C01822=1224.483,329.807,-70.540,-176.134,7.147,148.210
C01823=1224.479,330.055,-70.571,-176.132,7.149,148.210
C01824=1224.475,330.303,-70.602,-176.130,7.152,148.210
C01825=1224.470,330.551,-70.633,-176.128,7.155,148.211
C01826=1224.466,330.798,-70.664,-176.126,7.157,148.211
C01827=1224.462,331.047,-70.695,-176.124,7.160,148.211
C01828=1224.458,331.294,-70.727,-176.121,7.163,148.211
C01829=1224.454,331.543,-70.758,-176.120,7.165,148.211
C01830=1224.449,331.791,-70.789,-176.117,7.168,148.211
C01831=1224.445,332.039,-70.820,-176.115,7.171,148.211
C01832=1224.441,332.287,-70.851,-176.113,7.173,148.211
C01833=1224.436,332.535,-70.882,-176.111,7.176,148.211
C01834=1224.432,332.783,-70.914,-176.109,7.179,148.211
C01835=1224.428,333.031,-70.945,-176.107,7.181,148.211
C01836=1224.424,333.279,-70.976,-176.105,7.184,148.212
C01837=1224.419,333.527,-71.007,-176.103,7.187,148.212
C01838=1224.415,333.776,-71.038,-176.101,7.189,148.212
C01839=1224.411,334.023,-71.070,-176.099,7.192,148.212
C01840=1224.406,334.271,-71.101,-176.097,7.195,148.212
C01841=1224.403,334.519,-71.132,-176.095,7.198,148.212
C01842=1224.398,334.767,-71.163,-176.093,7.200,148.212
C01843=1224.394,335.015,-71.195,-176.091,7.203,148.212
C01844=1224.390,335.263,-71.226,-176.089,7.206,148.212
C01845=1224.386,335.511,-71.258,-176.087,7.209,148.213
C01846=1224.381,335.759,-71.288,-176.085,7.211,148.212
C01847=1224.378,336.007,-71.320,-176.083,7.214,148.213
C01848=1224.373,336.254,-71.352,-176.081,7.217,148.213
C01849=1224.369,336.503,-71.383,-176.079,7.219,148.213
C01850=1224.365,336.750,-71.414,-176.077,7.222,148.213
C01851=1224.361,336.999,-71.445,-176.075,7.225,148.213
C01852=1224.356,337.247,-71.478,-176.073,7.227,148.213
C01853=1224.352,337.495,-71.509,-176.071,7.230,148.213
C01854=1224.348,337.743,-71.540,-176.069,7.233,148.214
C01855=1224.344,337.991,-71.572,-176.067,7.235,148.214
C01856=1224.339,338.239,-71.603,-176.065,7.238,148.214
C01857=1224.336,338.487,-71.635,-176.063,7.241,148.214
C01858=1224.331,338.734,-71.666,-176.061,7.243,148.214
C01859=1224.327,338.983,-71.697,-176.059,7.247,148.214
C01860=1224.323,339.231,-71.730,-176.057,7.249,148.214
C01861=1224.319,339.478,-71.761,-176.055,7.251,148.214
C01862=1224.315,339.727,-71.792,-176.053,7.255,148.215
C01863=1224.310,339.974,-71.824,-176.051,7.257,148.215
C01864=1224.307,340.222,-71.856,-176.049,7.261,148.215
C01865=1224.302,340.470,-71.888,-176.047,7.263,148.215
C01866=1224.298,340.719,-71.919,-176.046,7.265,148.215
C01867=1224.293,340.996,-71.954,-176.043,7.269,148.215
C01868=1224.289,341.274,-71.990,-176.041,7.272,148.216
C01869=1224.283,341.552,-72.025,-176.039,7.274,148.216
C01870=1224.279,341.829,-72.061,-176.037,7.278,148.216
C01871=1224.275,342.077,-72.093,-176.035,7.280,148.216
C01872=1224.271,342.325,-72.124,-176.033,7.284,148.216
C01873=1224.266,342.573,-72.156,-176.031,7.286,148.216
C01874=1224.262,342.821,-72.188,-176.029,7.288,148.216
C01875=1224.258,343.069,-72.219,-176.027,7.292,148.217
C01876=1224.253,343.317,-72.252,-176.026,7.294,148.217
C01877=1224.250,343.565,-72.283,-176.024,7.297,148.217
C01878=1224.245,343.813,-72.315,-176.022,7.300,148.217
C01879=1224.242,344.061,-72.347,-176.020,7.302,148.217
C01880=1224.237,344.308,-72.379,-176.018,7.305,148.217
C01881=1224.233,344.557,-72.410,-176.016,7.308,148.218
C01882=1224.229,344.805,-72.442,-176.014,7.311,148.218
C01883=1224.224,345.053,-72.474,-176.013,7.313,148.218
C01884=1224.220,345.301,-72.506,-176.010,7.317,148.218
C01885=1224.216,345.549,-72.538,-176.009,7.319,148.218
C01886=1224.211,345.796,-72.570,-176.007,7.322,148.218
C01887=1224.208,346.044,-72.601,-176.005,7.325,148.219
C01888=1224.203,346.292,-72.634,-176.003,7.327,148.219
C01889=1224.199,346.540,-72.665,-176.001,7.330,148.219
C01890=1224.195,346.788,-72.697,-175.999,7.333,148.219
C01891=1224.190,347.036,-72.729,-175.997,7.336,148.219
C01892=1224.186,347.284,-72.761,-175.996,7.338,148.219
C01893=1224.182,347.532,-72.794,-175.994,7.341,148.220
C01894=1224.178,347.779,-72.825,-175.992,7.344,148.220
C01895=1224.174,348.027,-72.857,-175.990,7.347,148.220
C01896=1224.170,348.276,-72.889,-175.989,7.349,148.220
C01897=1224.166,348.523,-72.922,-175.987,7.352,148.220
C01898=1224.161,348.771,-72.954,-175.985,7.355,148.221
C01899=1224.157,349.019,-72.986,-175.983,7.357,148.221
C01900=1224.153,349.267,-73.018,-175.981,7.361,148.221
C01901=1224.149,349.515,-73.050,-175.979,7.363,148.221
C01902=1224.144,349.763,-73.082,-175.978,7.366,148.221
C01903=1224.141,350.011,-73.114,-175.976,7.368,148.222
C01904=1224.136,350.258,-73.146,-175.974,7.372,148.222
C01905=1224.132,350.506,-73.179,-175.972,7.374,148.222
C01906=1224.128,350.754,-73.211,-175.971,7.377,148.222
C01907=1224.124,351.002,-73.243,-175.969,7.380,148.222
C01908=1224.120,351.250,-73.274,-175.967,7.383,148.223
C01909=1224.115,351.498,-73.307,-175.965,7.385,148.223
C01910=1224.112,351.746,-73.339,-175.964,7.388,148.223
C01911=1224.107,351.994,-73.372,-175.961,7.391,148.223
C01912=1224.102,352.242,-73.404,-175.960,7.394,148.223
C01913=1224.099,352.490,-73.436,-175.959,7.397,148.224
C01914=1224.094,352.737,-73.469,-175.957,7.399,148.224
C01915=1224.091,352.985,-73.501,-175.955,7.402,148.224
C01916=1224.086,353.233,-73.533,-175.953,7.405,148.224
C01917=1224.082,353.481,-73.565,-175.952,7.407,148.225
C01918=1224.078,353.729,-73.598,-175.949,7.411,148.225
C01919=1224.074,353.977,-73.630,-175.948,7.413,148.225
C01920=1224.070,354.225,-73.662,-175.946,7.416,148.225
C01921=1224.065,354.472,-73.695,-175.945,7.419,148.226
C01922=1224.061,354.720,-73.727,-175.943,7.422,148.226
C01923=1224.057,354.969,-73.759,-175.941,7.425,148.226
C01924=1224.053,355.216,-73.792,-175.940,7.427,148.226
C01925=1224.049,355.464,-73.824,-175.938,7.430,148.226
C01926=1224.044,355.711,-73.857,-175.936,7.433,148.227
C01927=1224.041,355.959,-73.889,-175.935,7.436,148.227
C01928=1224.036,356.208,-73.921,-175.933,7.438,148.227
C01929=1224.032,356.455,-73.954,-175.931,7.441,148.227
C01930=1224.028,356.704,-73.986,-175.929,7.444,148.228
C01931=1224.024,356.951,-74.019,-175.928,7.447,148.228
C01932=1224.020,357.199,-74.051,-175.926,7.450,148.228
C01933=1224.016,357.446,-74.084,-175.925,7.452,148.228
C01934=1224.011,357.695,-74.117,-175.923,7.455,148.229
C01935=1224.008,357.942,-74.149,-175.921,7.458,148.229
C01936=1224.003,358.190,-74.182,-175.920,7.461,148.229
C01937=1223.999,358.437,-74.214,-175.918,7.463,148.229
C01938=1223.994,358.686,-74.247,-175.916,7.466,148.230
C01939=1223.991,358.933,-74.279,-175.915,7.470,148.230
C01940=1223.986,359.182,-74.312,-175.913,7.472,148.230
C01941=1223.982,359.429,-74.345,-175.911,7.475,148.230
C01942=1223.979,359.677,-74.377,-175.910,7.477,148.231
C01943=1223.974,359.925,-74.410,-175.909,7.480,148.231
C01944=1223.970,360.173,-74.442,-175.906,7.483,148.231
C01945=1223.965,360.420,-74.475,-175.905,7.486,148.232
C01946=1223.961,360.669,-74.507,-175.904,7.489,148.232
C01947=1223.957,360.916,-74.540,-175.902,7.491,148.232
C01948=1223.953,361.164,-74.573,-175.901,7.494,148.232
C01949=1223.949,361.412,-74.606,-175.899,7.497,148.233
C01950=1223.945,361.660,-74.638,-175.897,7.500,148.233
C01951=1223.941,361.907,-74.671,-175.896,7.503,148.233
C01952=1223.937,362.156,-74.704,-175.894,7.505,148.233
C01953=1223.933,362.404,-74.737,-175.893,7.508,148.234
C01954=1223.929,362.651,-74.770,-175.891,7.511,148.234
C01955=1223.924,362.899,-74.802,-175.890,7.514,148.234
C01956=1223.920,363.146,-74.835,-175.888,7.517,148.235
C01957=1223.916,363.394,-74.868,-175.887,7.520,148.235
C01958=1223.911,363.642,-74.900,-175.885,7.522,148.235
C01959=1223.907,363.890,-74.934,-175.884,7.525,148.236
C01960=1223.904,364.138,-74.966,-175.882,7.528,148.236
C01961=1223.900,364.385,-74.999,-175.881,7.531,148.236
C01962=1223.895,364.634,-75.032,-175.879,7.534,148.236
C01963=1223.891,364.881,-75.065,-175.878,7.536,148.237
C01964=1223.887,365.129,-75.098,-175.876,7.539,148.237
C01965=1223.883,365.377,-75.131,-175.875,7.542,148.237
C01966=1223.879,365.625,-75.163,-175.873,7.544,148.237
C01967=1223.875,365.873,-75.196,-175.872,7.547,148.238
C01968=1223.871,366.120,-75.229,-175.870,7.551,148.238
C01969=1223.867,366.368,-75.263,-175.869,7.553,148.239
C01970=1223.863,366.616,-75.296,-175.867,7.556,148.239
C01971=1223.858,366.896,-75.333,-175.866,7.559,148.239
C01972=1223.853,367.176,-75.370,-175.864,7.562,148.240
C01973=1223.849,367.455,-75.408,-175.863,7.565,148.240
C01974=1223.844,367.735,-75.444,-175.861,7.569,148.240
C01975=1223.840,367.983,-75.478,-175.860,7.571,148.241
C01976=1223.836,368.231,-75.510,-175.858,7.574,148.241
C01977=1223.832,368.478,-75.543,-175.857,7.577,148.241
C01978=1223.828,368.726,-75.576,-175.856,7.580,148.242
C01979=1223.824,368.974,-75.610,-175.854,7.582,148.242
C01980=1223.820,369.221,-75.643,-175.853,7.585,148.242
C01981=1223.815,369.469,-75.676,-175.852,7.588,148.243
C01982=1223.811,369.717,-75.709,-175.850,7.590,148.243
C01983=1223.807,369.965,-75.742,-175.849,7.593,148.243
C01984=1223.803,370.212,-75.775,-175.848,7.596,148.244
C01985=1223.799,370.461,-75.808,-175.846,7.598,148.244
C01986=1223.794,370.708,-75.841,-175.845,7.602,148.244
C01987=1223.790,370.956,-75.874,-175.843,7.605,148.245
C01988=1223.786,371.204,-75.907,-175.842,7.607,148.245
C01989=1223.782,371.452,-75.940,-175.841,7.610,148.245
C01990=1223.778,371.699,-75.974,-175.839,7.613,148.246
C01991=1223.774,371.947,-76.007,-175.838,7.616,148.246
C01992=1223.770,372.194,-76.041,-175.837,7.618,148.246
C01993=1223.766,372.442,-76.074,-175.835,7.621,148.247
C01994=1223.762,372.690,-76.107,-175.834,7.624,148.247
C01995=1223.758,372.937,-76.140,-175.833,7.627,148.247
C01996=1223.753,373.185,-76.173,-175.832,7.630,148.248
C01997=1223.748,373.433,-76.207,-175.830,7.632,148.248
C01998=1223.744,373.681,-76.240,-175.829,7.635,148.248
C01999=1223.740,373.929,-76.273,-175.828,7.637,148.249
C02000=1223.736,374.176,-76.306,-175.827,7.640,148.249
C02001=1223.733,374.425,-76.340,-175.826,7.643,148.249
C02002=1223.728,374.672,-76.373,-175.825,7.645,148.250
C02003=1223.724,374.920,-76.406,-175.823,7.648,148.250
C02004=1223.720,375.167,-76.440,-175.822,7.651,148.250
C02005=1223.716,375.415,-76.473,-175.821,7.654,148.251
C02006=1223.712,375.663,-76.506,-175.820,7.656,148.251
C02007=1223.708,375.911,-76.540,-175.819,7.659,148.252
C02008=1223.704,376.158,-76.573,-175.817,7.662,148.252
C02009=1223.699,376.406,-76.607,-175.816,7.665,148.252
C02010=1223.695,376.653,-76.640,-175.815,7.668,148.253
C02011=1223.692,376.902,-76.674,-175.813,7.670,148.253
C02012=1223.687,377.150,-76.707,-175.812,7.673,148.253
C02013=1223.683,377.397,-76.740,-175.812,7.675,148.254
C02014=1223.679,377.645,-76.773,-175.810,7.678,148.254
C02015=1223.675,377.892,-76.807,-175.809,7.681,148.255
C02016=1223.671,378.140,-76.841,-175.808,7.684,148.255
C02017=1223.666,378.388,-76.874,-175.807,7.686,148.255
C02018=1223.662,378.636,-76.907,-175.806,7.689,148.256
C02019=1223.658,378.883,-76.941,-175.805,7.692,148.256
C02020=1223.655,379.131,-76.975,-175.803,7.695,148.257
C02021=1223.651,379.379,-77.008,-175.803,7.697,148.257
C02022=1223.646,379.626,-77.042,-175.802,7.700,148.257
C02023=1223.642,379.874,-77.075,-175.800,7.702,148.258
C02024=1223.638,380.122,-77.109,-175.799,7.705,148.258
C02025=1223.634,380.369,-77.142,-175.798,7.708,148.258
C02026=1223.629,380.617,-77.176,-175.797,7.711,148.259
C02027=1223.626,380.865,-77.210,-175.796,7.713,148.259
C02028=1223.622,381.113,-77.243,-175.795,7.716,148.260
C02029=1223.618,381.360,-77.277,-175.794,7.719,148.260
C02030=1223.614,381.608,-77.310,-175.793,7.721,148.260
C02031=1223.609,381.855,-77.344,-175.792,7.724,148.261
C02032=1223.605,382.103,-77.378,-175.791,7.726,148.261
C02033=1223.601,382.351,-77.411,-175.790,7.729,148.261
C02034=1223.597,382.599,-77.445,-175.789,7.732,148.262
C02035=1223.593,382.847,-77.479,-175.788,7.735,148.262
C02036=1223.588,383.094,-77.512,-175.787,7.737,148.263
C02037=1223.585,383.341,-77.546,-175.786,7.740,148.263
C02038=1223.580,383.590,-77.580,-175.785,7.743,148.264
C02039=1223.577,383.837,-77.614,-175.784,7.745,148.264
C02040=1223.572,384.085,-77.647,-175.783,7.747,148.264
C02041=1223.569,384.332,-77.681,-175.782,7.750,148.265
C02042=1223.564,384.580,-77.715,-175.781,7.753,148.265
C02043=1223.560,384.828,-77.749,-175.780,7.756,148.266
C02044=1223.556,385.076,-77.782,-175.779,7.758,148.266
C02045=1223.551,385.324,-77.816,-175.778,7.761,148.267
C02046=1223.548,385.571,-77.850,-175.777,7.764,148.267
C02047=1223.543,385.819,-77.883,-175.776,7.766,148.267
C02048=1223.539,386.067,-77.918,-175.775,7.768,148.268
C02049=1223.535,386.314,-77.951,-175.774,7.771,148.268
C02050=1223.532,386.562,-77.985,-175.773,7.774,148.268
C02051=1223.527,386.809,-78.019,-175.773,7.776,148.269
C02052=1223.523,387.057,-78.052,-175.771,7.779,148.269
C02053=1223.520,387.305,-78.086,-175.770,7.782,148.270
C02054=1223.515,387.553,-78.120,-175.770,7.784,148.270
C02055=1223.511,387.800,-78.154,-175.768,7.787,148.271
C02056=1223.507,388.047,-78.187,-175.768,7.790,148.271
C02057=1223.503,388.296,-78.222,-175.767,7.792,148.271
C02058=1223.499,388.543,-78.255,-175.766,7.795,148.272
C02059=1223.495,388.790,-78.289,-175.765,7.798,148.272
C02060=1223.490,389.038,-78.324,-175.764,7.800,148.273
C02061=1223.487,389.286,-78.357,-175.763,7.803,148.273
C02062=1223.482,389.534,-78.392,-175.763,7.805,148.274
C02063=1223.478,389.781,-78.425,-175.762,7.807,148.274
C02064=1223.474,390.028,-78.459,-175.760,7.810,148.274
C02065=1223.470,390.277,-78.493,-175.760,7.812,148.275
C02066=1223.466,390.524,-78.527,-175.759,7.815,148.275
C02067=1223.461,390.772,-78.561,-175.758,7.817,148.276
C02068=1223.458,391.020,-78.595,-175.757,7.820,148.276
C02069=1223.454,391.267,-78.628,-175.756,7.823,148.276
C02070=1223.450,391.515,-78.663,-175.756,7.825,148.277
C02071=1223.446,391.762,-78.697,-175.755,7.828,148.277
C02072=1223.441,392.011,-78.731,-175.754,7.830,148.278
C02073=1223.438,392.258,-78.765,-175.753,7.833,148.278
C02074=1223.433,392.505,-78.799,-175.753,7.835,148.279
C02075=1223.429,392.787,-78.837,-175.752,7.838,148.279
C02076=1223.424,393.068,-78.876,-175.751,7.841,148.280
C02077=1223.419,393.351,-78.915,-175.750,7.844,148.280
C02078=1223.415,393.632,-78.954,-175.749,7.847,148.281
C02079=1223.411,393.879,-78.988,-175.748,7.849,148.281
C02080=1223.406,394.127,-79.021,-175.747,7.852,148.281
C02081=1223.402,394.375,-79.056,-175.746,7.854,148.282
C02082=1223.399,394.622,-79.090,-175.746,7.857,148.282
C02083=1223.394,394.870,-79.125,-175.745,7.859,148.283
C02084=1223.390,395.118,-79.158,-175.744,7.862,148.283
C02085=1223.386,395.366,-79.193,-175.744,7.864,148.284
C02086=1223.382,395.613,-79.226,-175.743,7.867,148.284
C02087=1223.378,395.861,-79.261,-175.742,7.869,148.284
C02088=1223.374,396.109,-79.294,-175.741,7.872,148.285
C02089=1223.369,396.356,-79.329,-175.741,7.874,148.285
C02090=1223.366,396.604,-79.363,-175.739,7.877,148.286
C02091=1223.362,396.851,-79.398,-175.739,7.879,148.286
C02092=1223.358,397.098,-79.431,-175.738,7.882,148.287
C02093=1223.354,397.346,-79.466,-175.737,7.884,148.287
C02094=1223.350,397.594,-79.499,-175.737,7.886,148.288
C02095=1223.345,397.842,-79.534,-175.736,7.889,148.288
C02096=1223.342,398.089,-79.568,-175.735,7.891,148.288
C02097=1223.337,398.337,-79.603,-175.735,7.894,148.289
C02098=1223.333,398.584,-79.636,-175.734,7.896,148.289
C02099=1223.329,398.832,-79.671,-175.733,7.898,148.290
C02100=1223.325,399.080,-79.705,-175.733,7.901,148.290
C02101=1223.321,399.327,-79.739,-175.732,7.903,148.290
C02102=1223.317,399.575,-79.774,-175.731,7.906,148.291
C02103=1223.313,399.822,-79.808,-175.731,7.908,148.291
C02104=1223.309,400.071,-79.842,-175.730,7.910,148.292
C02105=1223.305,400.318,-79.876,-175.729,7.913,148.292
C02106=1223.301,400.565,-79.911,-175.729,7.915,148.293
C02107=1223.297,400.813,-79.946,-175.728,7.917,148.293
C02108=1223.293,401.060,-79.980,-175.727,7.920,148.294
C02109=1223.288,401.308,-80.014,-175.727,7.922,148.294
C02110=1223.285,401.556,-80.048,-175.725,7.925,148.294
C02111=1223.280,401.803,-80.083,-175.725,7.927,148.295
C02112=1223.276,402.052,-80.117,-175.725,7.929,148.295
C02113=1223.272,402.299,-80.151,-175.723,7.932,148.296
C02114=1223.268,402.546,-80.185,-175.723,7.934,148.296
C02115=1223.265,402.794,-80.219,-175.723,7.936,148.297
C02116=1223.260,403.041,-80.254,-175.722,7.939,148.297
C02117=1223.256,403.290,-80.289,-175.721,7.941,148.297
C02118=1223.252,403.537,-80.323,-175.721,7.943,148.298
C02119=1223.248,403.784,-80.357,-175.720,7.946,148.298
C02120=1223.244,404.032,-80.392,-175.719,7.949,148.299
C02121=1223.240,404.279,-80.426,-175.719,7.950,148.299
C02122=1223.236,404.527,-80.461,-175.718,7.953,148.300
C02123=1223.231,404.775,-80.495,-175.718,7.955,148.300
C02124=1223.227,405.022,-80.529,-175.717,7.958,148.301
C02125=1223.223,405.270,-80.564,-175.716,7.960,148.301
C02126=1223.219,405.518,-80.598,-175.716,7.962,148.301
C02127=1223.216,405.765,-80.633,-175.715,7.965,148.302
C02128=1223.211,406.012,-80.668,-175.714,7.967,148.302
C02129=1223.207,406.260,-80.702,-175.714,7.969,148.303
C02130=1223.204,406.507,-80.736,-175.714,7.971,148.303
C02131=1223.199,406.755,-80.771,-175.712,7.974,148.303
C02132=1223.195,407.003,-80.806,-175.712,7.976,148.304
C02133=1223.191,407.250,-80.839,-175.712,7.978,148.304
C02134=1223.187,407.498,-80.874,-175.711,7.980,148.305
C02135=1223.183,407.746,-80.909,-175.711,7.982,148.305
C02136=1223.179,407.993,-80.943,-175.710,7.985,148.306
C02137=1223.175,408.241,-80.977,-175.709,7.988,148.306
C02138=1223.170,408.488,-81.012,-175.709,7.990,148.307
C02139=1223.167,408.736,-81.047,-175.708,7.992,148.307
C02140=1223.163,408.983,-81.081,-175.708,7.994,148.307
C02141=1223.159,409.231,-81.116,-175.707,7.997,148.308
C02142=1223.154,409.478,-81.151,-175.707,7.999,148.308
C02143=1223.151,409.726,-81.185,-175.706,8.001,148.309
C02144=1223.146,409.974,-81.219,-175.705,8.003,148.309
C02145=1223.143,410.222,-81.254,-175.705,8.005,148.310
C02146=1223.138,410.468,-81.289,-175.704,8.008,148.310
C02147=1223.135,410.716,-81.324,-175.704,8.010,148.311
C02148=1223.130,410.964,-81.358,-175.703,8.012,148.311
C02149=1223.126,411.211,-81.393,-175.702,8.014,148.311
C02150=1223.122,411.459,-81.427,-175.702,8.016,148.312
C02151=1223.118,411.706,-81.461,-175.702,8.018,148.312
C02152=1223.114,411.954,-81.497,-175.701,8.020,148.312
C02153=1223.110,412.201,-81.531,-175.700,8.023,148.313
C02154=1223.106,412.449,-81.566,-175.700,8.025,148.313
C02155=1223.102,412.697,-81.600,-175.699,8.028,148.314
C02156=1223.098,412.945,-81.635,-175.699,8.030,148.314
C02157=1223.094,413.191,-81.670,-175.698,8.032,148.315
C02158=1223.090,413.440,-81.705,-175.698,8.034,148.315
C02159=1223.086,413.687,-81.739,-175.697,8.036,148.315
C02160=1223.082,413.935,-81.774,-175.697,8.038,148.316
C02161=1223.078,414.182,-81.809,-175.696,8.041,148.316
C02162=1223.074,414.430,-81.844,-175.695,8.043,148.317
C02163=1223.069,414.677,-81.878,-175.695,8.045,148.317
C02164=1223.066,414.925,-81.912,-175.694,8.047,148.318
C02165=1223.062,415.172,-81.947,-175.694,8.049,148.318
C02166=1223.058,415.420,-81.982,-175.694,8.051,148.318
C02167=1223.051,415.838,-82.041,-175.692,8.055,148.319
C02168=1223.043,416.255,-82.099,-175.692,8.059,148.320
C02169=1223.037,416.673,-82.158,-175.691,8.063,148.321
C02170=1223.033,417.091,-82.216,-175.690,8.066,148.321
C02171=1222.612,417.091,-82.251,-175.693,8.076,148.325
C02172=1222.612,416.881,-82.221,-175.694,8.074,148.324
C02173=1222.615,416.671,-82.192,-175.694,8.073,148.324
C02174=1222.619,416.460,-82.162,-175.694,8.071,148.324
C02175=1222.622,416.250,-82.133,-175.695,8.069,148.324
C02176=1222.626,416.040,-82.103,-175.696,8.067,148.323
C02177=1222.628,415.830,-82.073,-175.696,8.065,148.323
C02178=1222.633,415.620,-82.044,-175.696,8.064,148.322
C02179=1222.635,415.409,-82.015,-175.697,8.062,148.322
C02180=1222.640,415.162,-81.980,-175.697,8.060,148.322
C02181=1222.644,414.914,-81.945,-175.697,8.058,148.321
C02182=1222.647,414.667,-81.911,-175.698,8.056,148.321
C02183=1222.651,414.419,-81.876,-175.699,8.054,148.320
C02184=1222.656,414.171,-81.841,-175.699,8.050,148.320
C02185=1222.660,413.924,-81.806,-175.700,8.049,148.320
C02186=1222.664,413.676,-81.771,-175.701,8.047,148.319
C02187=1222.667,413.429,-81.737,-175.701,8.044,148.319
C02188=1222.672,413.181,-81.703,-175.702,8.042,148.318
C02189=1222.676,412.934,-81.667,-175.702,8.040,148.318
C02190=1222.680,412.686,-81.633,-175.702,8.038,148.317
C02191=1222.684,412.438,-81.598,-175.703,8.036,148.317
C02192=1222.688,412.191,-81.564,-175.703,8.034,148.317
C02193=1222.692,411.943,-81.529,-175.704,8.031,148.316
C02194=1222.696,411.696,-81.494,-175.705,8.029,148.316
C02195=1222.700,411.448,-81.459,-175.705,8.027,148.315
C02196=1222.704,411.201,-81.425,-175.706,8.025,148.315
C02197=1222.709,410.954,-81.391,-175.706,8.022,148.314
C02198=1222.713,410.705,-81.356,-175.707,8.021,148.314
C02199=1222.717,410.459,-81.321,-175.708,8.018,148.314
C02200=1222.720,410.211,-81.286,-175.708,8.015,148.313
C02201=1222.725,409.963,-81.252,-175.709,8.013,148.313
C02202=1222.729,409.715,-81.217,-175.709,8.011,148.312
C02203=1222.733,409.468,-81.183,-175.710,8.009,148.312
C02204=1222.736,409.220,-81.148,-175.710,8.007,148.312
C02205=1222.741,408.973,-81.113,-175.711,8.004,148.311
C02206=1222.745,408.725,-81.078,-175.712,8.002,148.311
C02207=1222.749,408.478,-81.045,-175.712,8.000,148.310
C02208=1222.752,408.230,-81.010,-175.712,7.998,148.310
C02209=1222.757,407.982,-80.975,-175.713,7.996,148.309
C02210=1222.762,407.735,-80.941,-175.714,7.993,148.309
C02211=1222.765,407.487,-80.907,-175.714,7.991,148.308
C02212=1222.769,407.240,-80.872,-175.715,7.989,148.308
C02213=1222.773,406.992,-80.837,-175.715,7.987,148.308
C02214=1222.777,406.745,-80.803,-175.716,7.985,148.307
C02215=1222.781,406.497,-80.768,-175.717,7.981,148.307
C02216=1222.785,406.250,-80.733,-175.717,7.980,148.306
C02217=1222.789,406.003,-80.700,-175.717,7.977,148.306
C02218=1222.793,405.754,-80.665,-175.718,7.975,148.305
C02219=1222.798,405.507,-80.630,-175.719,7.972,148.305
C02220=1222.801,405.259,-80.596,-175.719,7.970,148.305
C02221=1222.806,405.012,-80.562,-175.720,7.968,148.304
C02222=1222.810,404.764,-80.527,-175.721,7.965,148.304
C02223=1222.813,404.517,-80.493,-175.721,7.963,148.303
C02224=1222.818,404.269,-80.458,-175.722,7.961,148.303
C02225=1222.822,404.021,-80.424,-175.722,7.959,148.302
C02226=1222.826,403.774,-80.390,-175.723,7.956,148.302
C02227=1222.830,403.526,-80.355,-175.724,7.954,148.301
C02228=1222.834,403.278,-80.320,-175.724,7.952,148.301
C02229=1222.838,403.031,-80.286,-175.725,7.949,148.301
C02230=1222.842,402.783,-80.252,-175.726,7.947,148.300
C02231=1222.847,402.536,-80.217,-175.726,7.945,148.300
C02232=1222.850,402.288,-80.183,-175.727,7.943,148.299
C02233=1222.855,402.040,-80.148,-175.728,7.940,148.299
C02234=1222.858,401.793,-80.115,-175.728,7.938,148.299
C02235=1222.862,401.545,-80.080,-175.728,7.935,148.298
C02236=1222.867,401.298,-80.045,-175.730,7.933,148.298
C02237=1222.870,401.050,-80.011,-175.730,7.931,148.297
C02238=1222.875,400.803,-79.977,-175.731,7.927,148.297
C02239=1222.879,400.555,-79.943,-175.732,7.926,148.296
C02240=1222.882,400.307,-79.908,-175.732,7.924,148.296
C02241=1222.887,400.059,-79.874,-175.733,7.920,148.295
C02242=1222.891,399.812,-79.840,-175.734,7.918,148.295
C02243=1222.895,399.564,-79.805,-175.734,7.916,148.294
C02244=1222.899,399.317,-79.772,-175.735,7.913,148.294
C02245=1222.903,399.069,-79.737,-175.736,7.911,148.294
C02246=1222.908,398.821,-79.702,-175.736,7.908,148.293
C02247=1222.911,398.574,-79.668,-175.737,7.906,148.293
C02248=1222.915,398.326,-79.634,-175.738,7.904,148.292
C02249=1222.919,398.079,-79.600,-175.738,7.901,148.292
C02250=1222.924,397.831,-79.566,-175.739,7.899,148.292
C02251=1222.927,397.583,-79.532,-175.740,7.896,148.291
C02252=1222.932,397.336,-79.497,-175.740,7.894,148.291
C02253=1222.936,397.089,-79.463,-175.741,7.892,148.290
C02254=1222.940,396.841,-79.429,-175.742,7.889,148.290
C02255=1222.943,396.593,-79.395,-175.742,7.887,148.289
C02256=1222.948,396.345,-79.361,-175.744,7.884,148.289
C02257=1222.952,396.097,-79.326,-175.744,7.882,148.289
C02258=1222.956,395.850,-79.292,-175.745,7.879,148.288
C02259=1222.961,395.603,-79.258,-175.746,7.877,148.288
C02260=1222.964,395.355,-79.224,-175.747,7.874,148.287
C02261=1222.969,395.107,-79.190,-175.747,7.872,148.287
C02262=1222.973,394.860,-79.156,-175.748,7.869,148.286
C02263=1222.977,394.612,-79.121,-175.749,7.867,148.286
C02264=1222.980,394.365,-79.087,-175.749,7.864,148.285
C02265=1222.985,394.117,-79.053,-175.750,7.862,148.285
C02266=1222.989,393.869,-79.019,-175.751,7.859,148.285
C02267=1222.992,393.622,-78.985,-175.751,7.857,148.284
C02268=1222.997,393.340,-78.946,-175.753,7.854,148.284
C02269=1223.002,393.058,-78.908,-175.753,7.851,148.283
C02270=1223.007,392.776,-78.868,-175.755,7.848,148.283
C02271=1223.011,392.494,-78.830,-175.755,7.845,148.282
C02272=1223.016,392.247,-78.796,-175.756,7.843,148.282
C02273=1223.019,392.000,-78.762,-175.757,7.840,148.281
C02274=1223.024,391.752,-78.729,-175.758,7.838,148.281
C02275=1223.028,391.504,-78.694,-175.758,7.835,148.280
C02276=1223.031,391.257,-78.660,-175.759,7.833,148.280
C02277=1223.036,391.009,-78.626,-175.760,7.831,148.280
C02278=1223.039,390.761,-78.592,-175.761,7.828,148.279
C02279=1223.044,390.514,-78.557,-175.762,7.825,148.279
C02280=1223.048,390.266,-78.524,-175.763,7.823,148.278
C02281=1223.052,390.019,-78.490,-175.763,7.821,148.278
C02282=1223.056,389.771,-78.456,-175.765,7.818,148.278
C02283=1223.060,389.523,-78.422,-175.765,7.815,148.277
C02284=1223.065,389.276,-78.388,-175.766,7.813,148.277
C02285=1223.069,389.028,-78.355,-175.767,7.810,148.276
C02286=1223.072,388.780,-78.321,-175.768,7.807,148.276
C02287=1223.077,388.533,-78.286,-175.769,7.805,148.275
C02288=1223.081,388.285,-78.253,-175.770,7.802,148.275
C02289=1223.085,388.038,-78.219,-175.770,7.800,148.275
C02290=1223.089,387.789,-78.185,-175.772,7.797,148.274
C02291=1223.093,387.542,-78.151,-175.773,7.794,148.274
C02292=1223.098,387.294,-78.117,-175.773,7.792,148.273
C02293=1223.101,387.047,-78.084,-175.774,7.789,148.273
C02294=1223.105,386.799,-78.049,-175.775,7.786,148.272
C02295=1223.110,386.551,-78.016,-175.776,7.784,148.272
C02296=1223.113,386.304,-77.982,-175.777,7.782,148.272
C02297=1223.118,386.056,-77.949,-175.778,7.779,148.271
C02298=1223.121,385.808,-77.914,-175.779,7.776,148.271
C02299=1223.126,385.560,-77.881,-175.780,7.774,148.270
C02300=1223.129,385.313,-77.847,-175.781,7.771,148.270
C02301=1223.134,385.065,-77.813,-175.782,7.768,148.269
C02302=1223.138,384.818,-77.779,-175.783,7.766,148.269
C02303=1223.142,384.570,-77.746,-175.784,7.763,148.269
C02304=1223.147,384.322,-77.712,-175.785,7.760,148.268
C02305=1223.150,384.074,-77.678,-175.786,7.757,148.268
C02306=1223.155,383.827,-77.645,-175.786,7.755,148.267
C02307=1223.158,383.580,-77.611,-175.787,7.753,148.267
C02308=1223.163,383.331,-77.577,-175.789,7.750,148.267
C02309=1223.166,383.084,-77.543,-175.790,7.747,148.266
C02310=1223.171,382.836,-77.510,-175.790,7.745,148.266
C02311=1223.174,382.589,-77.476,-175.792,7.742,148.265
C02312=1223.179,382.341,-77.442,-175.793,7.739,148.265
C02313=1223.183,382.092,-77.409,-175.794,7.736,148.265
C02314=1223.187,381.845,-77.375,-175.795,7.735,148.264
C02315=1223.192,381.597,-77.341,-175.796,7.732,148.264
C02316=1223.196,381.350,-77.308,-175.797,7.729,148.264
C02317=1223.200,381.102,-77.274,-175.798,7.726,148.263
C02318=1223.204,380.855,-77.241,-175.799,7.723,148.263
C02319=1223.207,380.606,-77.207,-175.800,7.720,148.262
C02320=1223.212,380.359,-77.173,-175.801,7.718,148.262
C02321=1223.216,380.111,-77.140,-175.802,7.715,148.261
C02322=1223.220,379.863,-77.106,-175.803,7.713,148.261
C02323=1223.224,379.616,-77.073,-175.804,7.710,148.261
C02324=1223.229,379.368,-77.039,-175.805,7.707,148.260
C02325=1223.233,379.121,-77.006,-175.807,7.704,148.260
C02326=1223.236,378.873,-76.971,-175.807,7.702,148.259
C02327=1223.240,378.625,-76.938,-175.808,7.699,148.259
C02328=1223.244,378.377,-76.905,-175.810,7.696,148.259
C02329=1223.249,378.130,-76.872,-175.811,7.694,148.258
C02330=1223.253,377.882,-76.838,-175.812,7.691,148.258
C02331=1223.257,377.634,-76.804,-175.814,7.688,148.258
C02332=1223.261,377.387,-76.771,-175.815,7.685,148.257
C02333=1223.266,377.139,-76.738,-175.816,7.683,148.257
C02334=1223.269,376.891,-76.704,-175.817,7.681,148.257
C02335=1223.273,376.643,-76.671,-175.818,7.678,148.256
C02336=1223.278,376.395,-76.637,-175.819,7.675,148.256
C02337=1223.282,376.148,-76.604,-175.820,7.672,148.255
C02338=1223.286,375.900,-76.571,-175.821,7.669,148.255
C02339=1223.290,375.653,-76.537,-175.822,7.667,148.255
C02340=1223.294,375.405,-76.504,-175.824,7.664,148.254
C02341=1223.298,375.157,-76.470,-175.825,7.661,148.254
C02342=1223.302,374.910,-76.437,-175.826,7.658,148.254
C02343=1223.306,374.662,-76.404,-175.828,7.656,148.253
C02344=1223.310,374.413,-76.371,-175.829,7.653,148.253
C02345=1223.314,374.166,-76.337,-175.830,7.650,148.252
C02346=1223.319,373.918,-76.303,-175.831,7.647,148.252
C02347=1223.323,373.671,-76.270,-175.832,7.644,148.252
C02348=1223.327,373.423,-76.237,-175.834,7.642,148.251
C02349=1223.331,373.175,-76.203,-175.835,7.639,148.251
C02350=1223.335,372.927,-76.170,-175.836,7.636,148.251
C02351=1223.339,372.680,-76.137,-175.837,7.633,148.250
C02352=1223.344,372.432,-76.104,-175.839,7.630,148.250
C02353=1223.348,372.184,-76.071,-175.840,7.628,148.250
C02354=1223.352,371.936,-76.038,-175.841,7.625,148.249
C02355=1223.356,371.689,-76.005,-175.843,7.622,148.249
C02356=1223.360,371.441,-75.971,-175.844,7.619,148.248
C02357=1223.364,371.193,-75.938,-175.845,7.617,148.248
C02358=1223.368,370.946,-75.905,-175.847,7.614,148.248
C02359=1223.372,370.698,-75.872,-175.848,7.611,148.248
C02360=1223.377,370.450,-75.839,-175.849,7.608,148.247
C02361=1223.381,370.202,-75.806,-175.851,7.606,148.247
C02362=1223.385,369.955,-75.772,-175.852,7.603,148.247
C02363=1223.388,369.706,-75.739,-175.853,7.600,148.246
C02364=1223.393,369.458,-75.706,-175.855,7.598,148.246
C02365=1223.397,369.211,-75.673,-175.856,7.595,148.246
C02366=1223.401,368.963,-75.639,-175.857,7.592,148.245
C02367=1223.405,368.715,-75.606,-175.859,7.590,148.245
C02368=1223.409,368.468,-75.573,-175.860,7.587,148.245
C02369=1223.413,368.220,-75.540,-175.861,7.584,148.244
C02370=1223.417,367.972,-75.507,-175.863,7.581,148.244
C02371=1223.422,367.724,-75.474,-175.864,7.578,148.244
C02372=1223.426,367.444,-75.437,-175.865,7.575,148.243
C02373=1223.431,367.165,-75.399,-175.868,7.572,148.243
C02374=1223.435,366.885,-75.362,-175.869,7.569,148.243
C02375=1223.440,366.605,-75.326,-175.871,7.565,148.242
C02376=1223.444,366.357,-75.292,-175.872,7.563,148.242
C02377=1223.449,366.110,-75.260,-175.873,7.560,148.241
C02378=1223.453,365.863,-75.226,-175.875,7.557,148.241
C02379=1223.457,365.614,-75.194,-175.876,7.554,148.241
C02380=1223.461,365.367,-75.161,-175.878,7.552,148.241
C02381=1223.466,365.119,-75.128,-175.879,7.549,148.240
C02382=1223.470,364.871,-75.095,-175.881,7.547,148.240
C02383=1223.473,364.624,-75.062,-175.882,7.543,148.240
C02384=1223.478,364.375,-75.030,-175.884,7.540,148.239
C02385=1223.482,364.128,-74.996,-175.885,7.538,148.239
C02386=1223.486,363.880,-74.963,-175.887,7.535,148.239
C02387=1223.490,363.632,-74.930,-175.888,7.532,148.239
C02388=1223.494,363.384,-74.898,-175.890,7.530,148.238
C02389=1223.498,363.136,-74.865,-175.891,7.526,148.238
C02390=1223.502,362.889,-74.832,-175.893,7.523,148.238
C02391=1223.506,362.640,-74.800,-175.894,7.521,148.237
C02392=1223.510,362.393,-74.766,-175.896,7.518,148.237
C02393=1223.515,362.145,-74.733,-175.897,7.515,148.237
C02394=1223.518,361.897,-74.701,-175.899,7.513,148.237
C02395=1223.523,361.650,-74.669,-175.901,7.509,148.236
C02396=1223.527,361.402,-74.635,-175.902,7.507,148.236
C02397=1223.532,361.154,-74.603,-175.904,7.504,148.236
C02398=1223.535,360.906,-74.570,-175.905,7.501,148.235
C02399=1223.539,360.659,-74.537,-175.906,7.499,148.235
C02400=1223.544,360.410,-74.505,-175.908,7.495,148.235
C02401=1223.548,360.162,-74.472,-175.910,7.493,148.234
C02402=1223.551,359.914,-74.440,-175.911,7.490,148.234
C02403=1223.556,359.667,-74.407,-175.913,7.487,148.234
C02404=1223.561,359.419,-74.375,-175.915,7.484,148.234
C02405=1223.565,359.171,-74.341,-175.916,7.481,148.233
C02406=1223.568,358.924,-74.309,-175.918,7.479,148.233
C02407=1223.573,358.676,-74.276,-175.919,7.476,148.233
C02408=1223.577,358.428,-74.243,-175.921,7.473,148.233
C02409=1223.580,358.180,-74.211,-175.923,7.470,148.232
C02410=1223.585,357.932,-74.178,-175.924,7.467,148.232
C02411=1223.590,357.684,-74.146,-175.926,7.465,148.232
C02412=1223.593,357.437,-74.114,-175.927,7.462,148.232
C02413=1223.598,357.189,-74.081,-175.930,7.459,148.231
C02414=1223.602,356.941,-74.048,-175.931,7.456,148.231
C02415=1223.605,356.693,-74.016,-175.932,7.453,148.231
C02416=1223.610,356.444,-73.984,-175.934,7.451,148.231
C02417=1223.615,356.197,-73.951,-175.936,7.448,148.230
C02418=1223.618,355.949,-73.919,-175.937,7.445,148.230
C02419=1223.622,355.702,-73.886,-175.939,7.442,148.230
C02420=1223.627,355.453,-73.854,-175.941,7.440,148.230
C02421=1223.631,355.205,-73.822,-175.943,7.436,148.230
C02422=1223.635,354.958,-73.789,-175.944,7.434,148.229
C02423=1223.639,354.710,-73.757,-175.946,7.431,148.229
C02424=1223.643,354.463,-73.724,-175.947,7.428,148.229
C02425=1223.648,354.214,-73.691,-175.949,7.425,148.229
C02426=1223.651,353.966,-73.660,-175.951,7.423,148.228
C02427=1223.656,353.719,-73.627,-175.953,7.420,148.228
C02428=1223.660,353.471,-73.595,-175.954,7.418,148.228
C02429=1223.664,353.223,-73.563,-175.956,7.414,148.228
C02430=1223.669,352.974,-73.530,-175.958,7.412,148.228
C02431=1223.672,352.727,-73.498,-175.959,7.409,148.227
C02432=1223.677,352.479,-73.465,-175.961,7.405,148.227
C02433=1223.681,352.231,-73.434,-175.963,7.403,148.227
C02434=1223.685,351.984,-73.400,-175.965,7.400,148.227
C02435=1223.689,351.735,-73.369,-175.966,7.398,148.226
C02436=1223.694,351.488,-73.337,-175.969,7.395,148.226
C02437=1223.697,351.240,-73.305,-175.970,7.392,148.226
C02438=1223.702,350.991,-73.272,-175.972,7.389,148.226
C02439=1223.705,350.744,-73.240,-175.974,7.386,148.226
C02440=1223.710,350.496,-73.208,-175.976,7.384,148.225
C02441=1223.714,350.248,-73.176,-175.977,7.381,148.225
C02442=1223.718,350.000,-73.143,-175.979,7.379,148.225
C02443=1223.723,349.753,-73.112,-175.981,7.375,148.225
C02444=1223.727,349.504,-73.079,-175.983,7.373,148.225
C02445=1223.731,349.257,-73.047,-175.984,7.370,148.224
C02446=1223.735,349.009,-73.014,-175.987,7.367,148.224
C02447=1223.739,348.761,-72.983,-175.988,7.364,148.224
C02448=1223.744,348.513,-72.950,-175.990,7.362,148.224
C02449=1223.747,348.265,-72.919,-175.992,7.358,148.224
C02450=1223.752,348.017,-72.887,-175.994,7.356,148.223
C02451=1223.756,347.769,-72.855,-175.995,7.353,148.223
C02452=1223.760,347.521,-72.823,-175.997,7.351,148.223
C02453=1223.765,347.273,-72.791,-175.999,7.347,148.223
C02454=1223.769,347.025,-72.759,-176.001,7.345,148.223
C02455=1223.772,346.777,-72.727,-176.002,7.342,148.222
C02456=1223.777,346.530,-72.695,-176.005,7.339,148.222
C02457=1223.781,346.282,-72.663,-176.006,7.336,148.222
C02458=1223.786,346.033,-72.631,-176.008,7.334,148.222
C02459=1223.790,345.786,-72.599,-176.010,7.331,148.222
C02460=1223.794,345.538,-72.567,-176.012,7.328,148.221
C02461=1223.798,345.290,-72.535,-176.014,7.326,148.221
C02462=1223.802,345.042,-72.504,-176.016,7.322,148.221
C02463=1223.806,344.794,-72.472,-176.018,7.320,148.221
C02464=1223.810,344.546,-72.439,-176.019,7.317,148.221
C02465=1223.815,344.299,-72.408,-176.021,7.314,148.221
C02466=1223.818,344.050,-72.376,-176.023,7.312,148.220
C02467=1223.824,343.803,-72.344,-176.025,7.309,148.220
C02468=1223.827,343.555,-72.312,-176.027,7.306,148.220
C02469=1223.831,343.307,-72.280,-176.029,7.303,148.220
C02470=1223.836,343.059,-72.248,-176.031,7.301,148.220
C02471=1223.840,342.810,-72.217,-176.033,7.298,148.220
C02472=1223.844,342.563,-72.185,-176.034,7.295,148.220
C02473=1223.848,342.315,-72.154,-176.036,7.292,148.219
C02474=1223.852,342.067,-72.121,-176.039,7.289,148.219
C02475=1223.857,341.819,-72.090,-176.040,7.287,148.219
C02476=1223.861,341.541,-72.055,-176.042,7.284,148.219
C02477=1223.866,341.263,-72.019,-176.044,7.281,148.219
C02478=1223.871,340.986,-71.983,-176.047,7.278,148.219
C02479=1223.875,340.708,-71.948,-176.049,7.275,148.218
C02480=1223.880,340.460,-71.917,-176.051,7.272,148.218
C02481=1223.884,340.212,-71.884,-176.053,7.269,148.218
C02482=1223.888,339.965,-71.853,-176.055,7.266,148.218
C02483=1223.892,339.716,-71.822,-176.056,7.264,148.218
C02484=1223.896,339.468,-71.790,-176.059,7.261,148.218
C02485=1223.900,339.221,-71.758,-176.060,7.258,148.218
C02486=1223.904,338.972,-71.727,-176.062,7.256,148.218
C02487=1223.910,338.724,-71.695,-176.065,7.252,148.217
C02488=1223.913,338.476,-71.663,-176.066,7.250,148.217
C02489=1223.918,338.228,-71.632,-176.068,7.248,148.217
C02490=1223.922,337.980,-71.601,-176.070,7.244,148.217
C02491=1223.926,337.733,-71.569,-176.072,7.242,148.217
C02492=1223.930,337.484,-71.538,-176.074,7.240,148.217
C02493=1223.934,337.237,-71.506,-176.076,7.236,148.217
C02494=1223.939,336.989,-71.474,-176.078,7.234,148.216
C02495=1223.943,336.741,-71.443,-176.080,7.232,148.216
C02496=1223.947,336.493,-71.411,-176.082,7.228,148.216
C02497=1223.952,336.245,-71.381,-176.084,7.226,148.216
C02498=1223.955,335.997,-71.349,-176.087,7.223,148.216
C02499=1223.960,335.749,-71.318,-176.088,7.220,148.216
C02500=1223.964,335.501,-71.286,-176.090,7.218,148.216
C02501=1223.968,335.253,-71.255,-176.092,7.214,148.216
C02502=1223.972,335.005,-71.224,-176.094,7.212,148.215
C02503=1223.977,334.757,-71.193,-176.096,7.210,148.216
C02504=1223.980,334.509,-71.161,-176.098,7.206,148.215
C02505=1223.985,334.261,-71.130,-176.100,7.204,148.215
C02506=1223.989,334.013,-71.098,-176.102,7.202,148.215
C02507=1223.993,333.765,-71.068,-176.104,7.198,148.215
C02508=1223.998,333.516,-71.035,-176.106,7.196,148.215
C02509=1224.002,333.268,-71.004,-176.109,7.193,148.215
C02510=1224.007,333.021,-70.973,-176.111,7.190,148.215
C02511=1224.011,332.772,-70.942,-176.112,7.188,148.215
C02512=1224.015,332.525,-70.910,-176.115,7.185,148.214
C02513=1224.019,332.276,-70.879,-176.117,7.182,148.214
C02514=1224.023,332.029,-70.849,-176.118,7.180,148.214
C02515=1224.026,331.781,-70.817,-176.121,7.177,148.214
C02516=1224.031,331.533,-70.786,-176.123,7.174,148.214
C02517=1224.036,331.285,-70.756,-176.125,7.172,148.214
C02518=1224.039,331.037,-70.724,-176.127,7.169,148.214
C02519=1224.044,330.789,-70.693,-176.129,7.166,148.214
C02520=1224.048,330.540,-70.662,-176.131,7.163,148.214
C02521=1224.052,330.293,-70.630,-176.133,7.161,148.214
C02522=1224.057,330.045,-70.600,-176.135,7.158,148.214
C02523=1224.061,329.796,-70.569,-176.137,7.155,148.214
C02524=1224.066,329.548,-70.538,-176.139,7.153,148.213
C02525=1224.069,329.300,-70.506,-176.141,7.150,148.213
C02526=1224.074,329.052,-70.475,-176.144,7.147,148.213
C02527=1224.078,328.804,-70.444,-176.146,7.145,148.213
C02528=1224.082,328.556,-70.414,-176.148,7.142,148.213
C02529=1224.086,328.309,-70.382,-176.150,7.139,148.213
C02530=1224.091,328.061,-70.352,-176.152,7.137,148.213
C02531=1224.095,327.812,-70.321,-176.154,7.134,148.213
C02532=1224.099,327.564,-70.290,-176.156,7.132,148.213
C02533=1224.103,327.315,-70.259,-176.158,7.129,148.213
C02534=1224.108,327.068,-70.227,-176.160,7.126,148.213
C02535=1224.111,326.820,-70.197,-176.163,7.124,148.213
C02536=1224.116,326.572,-70.166,-176.165,7.120,148.213
C02537=1224.120,326.324,-70.135,-176.167,7.118,148.213
C02538=1224.125,326.076,-70.104,-176.169,7.116,148.213
C02539=1224.129,325.827,-70.073,-176.171,7.113,148.212
C02540=1224.133,325.579,-70.043,-176.173,7.110,148.212
C02541=1224.137,325.332,-70.012,-176.175,7.108,148.212
C02542=1224.141,325.083,-69.981,-176.178,7.105,148.212
C02543=1224.146,324.836,-69.950,-176.180,7.103,148.212
C02544=1224.149,324.588,-69.919,-176.182,7.099,148.212
C02545=1224.154,324.340,-69.889,-176.184,7.097,148.212
C02546=1224.158,324.091,-69.858,-176.186,7.095,148.212
C02547=1224.163,323.843,-69.827,-176.188,7.091,148.212
C02548=1224.167,323.596,-69.797,-176.190,7.089,148.212
C02549=1224.171,323.347,-69.766,-176.192,7.087,148.212
C02550=1224.175,323.099,-69.735,-176.195,7.084,148.212
C02551=1224.179,322.851,-69.705,-176.197,7.081,148.212
C02552=1224.184,322.603,-69.674,-176.199,7.078,148.212
C02553=1224.188,322.354,-69.643,-176.201,7.076,148.212
C02554=1224.193,322.106,-69.613,-176.203,7.074,148.212
C02555=1224.196,321.859,-69.582,-176.206,7.070,148.212
C02556=1224.201,321.611,-69.552,-176.208,7.068,148.212
C02557=1224.205,321.362,-69.521,-176.210,7.066,148.212
C02558=1224.209,321.114,-69.490,-176.212,7.063,148.212
C02559=1224.214,320.866,-69.460,-176.214,7.060,148.212
C02560=1224.217,320.619,-69.429,-176.216,7.057,148.211
C02561=1224.221,320.370,-69.398,-176.219,7.055,148.212
C02562=1224.226,320.121,-69.368,-176.221,7.053,148.212
C02563=1224.230,319.874,-69.338,-176.223,7.050,148.212
C02564=1224.235,319.626,-69.307,-176.225,7.047,148.211
C02565=1224.239,319.378,-69.277,-176.227,7.045,148.211
C02566=1224.243,319.130,-69.246,-176.230,7.042,148.211
C02567=1224.248,318.881,-69.216,-176.232,7.040,148.211
C02568=1224.252,318.633,-69.186,-176.234,7.037,148.212
C02569=1224.256,318.385,-69.155,-176.236,7.034,148.211
C02570=1224.260,318.138,-69.125,-176.238,7.032,148.211
C02571=1224.264,317.889,-69.094,-176.241,7.029,148.211
C02572=1224.269,317.640,-69.064,-176.243,7.026,148.211
C02573=1224.273,317.393,-69.034,-176.245,7.024,148.211
C02574=1224.277,317.145,-69.003,-176.247,7.021,148.211
C02575=1224.282,316.897,-68.973,-176.249,7.019,148.211
C02576=1224.286,316.648,-68.942,-176.251,7.016,148.211
C02577=1224.290,316.400,-68.912,-176.254,7.013,148.211
C02578=1224.294,316.152,-68.882,-176.256,7.011,148.211
C02579=1224.298,315.904,-68.852,-176.258,7.008,148.211
C02580=1224.303,315.628,-68.818,-176.261,7.006,148.211
C02581=1224.307,315.352,-68.785,-176.263,7.003,148.211
C02582=1224.313,315.077,-68.751,-176.266,6.999,148.211
C02583=1224.318,314.801,-68.717,-176.268,6.996,148.211
C02584=1224.322,314.553,-68.687,-176.271,6.994,148.211
C02585=1224.326,314.305,-68.657,-176.273,6.992,148.211
C02586=1224.331,314.057,-68.627,-176.275,6.989,148.211
C02587=1224.334,313.808,-68.597,-176.277,6.987,148.211
C02588=1224.339,313.560,-68.566,-176.280,6.985,148.211
C02589=1224.343,313.312,-68.537,-176.282,6.981,148.211
C02590=1224.348,313.064,-68.506,-176.284,6.979,148.211
C02591=1224.352,312.815,-68.476,-176.286,6.977,148.211
C02592=1224.356,312.568,-68.446,-176.289,6.974,148.211
C02593=1224.361,312.319,-68.416,-176.291,6.971,148.211
C02594=1224.364,312.072,-68.386,-176.293,6.968,148.211
C02595=1224.369,311.823,-68.356,-176.296,6.966,148.211
C02596=1224.373,311.575,-68.326,-176.298,6.964,148.211
C02597=1224.377,311.327,-68.296,-176.300,6.961,148.211
C02598=1224.381,311.078,-68.265,-176.302,6.959,148.211
C02599=1224.386,310.830,-68.236,-176.304,6.956,148.212
C02600=1224.390,310.582,-68.206,-176.307,6.953,148.212
C02601=1224.394,310.334,-68.176,-176.309,6.951,148.212
C02602=1224.399,310.086,-68.146,-176.311,6.949,148.212
C02603=1224.402,309.838,-68.116,-176.314,6.946,148.212
C02604=1224.407,309.589,-68.086,-176.316,6.943,148.211
C02605=1224.412,309.341,-68.056,-176.318,6.941,148.212
C02606=1224.415,309.093,-68.026,-176.320,6.938,148.212
C02607=1224.420,308.845,-67.996,-176.323,6.936,148.212
C02608=1224.425,308.597,-67.967,-176.325,6.933,148.212
C02609=1224.428,308.349,-67.937,-176.327,6.931,148.212
C02610=1224.433,308.100,-67.907,-176.329,6.928,148.212
C02611=1224.438,307.852,-67.877,-176.332,6.925,148.212
C02612=1224.442,307.604,-67.848,-176.334,6.923,148.212
C02613=1224.446,307.356,-67.818,-176.336,6.921,148.212
C02614=1224.450,307.108,-67.787,-176.339,6.918,148.212
C02615=1224.455,306.859,-67.758,-176.341,6.916,148.212
C02616=1224.459,306.611,-67.729,-176.343,6.913,148.212
C02617=1224.463,306.363,-67.699,-176.346,6.910,148.212
C02618=1224.468,306.115,-67.668,-176.348,6.908,148.212
C02619=1224.472,305.867,-67.639,-176.350,6.906,148.212
C02620=1224.476,305.618,-67.609,-176.353,6.903,148.212
C02621=1224.480,305.370,-67.580,-176.355,6.901,148.212
C02622=1224.484,305.122,-67.551,-176.357,6.899,148.212
C02623=1224.489,304.874,-67.521,-176.360,6.896,148.212
C02624=1224.494,304.626,-67.491,-176.362,6.894,148.212
C02625=1224.498,304.378,-67.461,-176.364,6.891,148.212
C02626=1224.502,304.130,-67.432,-176.367,6.888,148.212
C02627=1224.506,303.881,-67.402,-176.369,6.886,148.213
C02628=1224.510,303.633,-67.373,-176.371,6.884,148.213
C02629=1224.515,303.385,-67.343,-176.374,6.881,148.213
C02630=1224.520,303.136,-67.313,-176.376,6.879,148.213
C02631=1224.524,302.888,-67.284,-176.378,6.876,148.213
C02632=1224.528,302.640,-67.254,-176.381,6.873,148.213
C02633=1224.532,302.392,-67.225,-176.383,6.871,148.213
C02634=1224.536,302.143,-67.196,-176.385,6.869,148.213
C02635=1224.541,301.896,-67.166,-176.388,6.866,148.213
C02636=1224.545,301.647,-67.137,-176.390,6.864,148.213
C02637=1224.549,301.399,-67.108,-176.392,6.862,148.213
C02638=1224.554,301.151,-67.078,-176.395,6.859,148.213
C02639=1224.558,300.903,-67.049,-176.397,6.856,148.213
C02640=1224.562,300.654,-67.019,-176.399,6.854,148.213
C02641=1224.566,300.406,-66.990,-176.402,6.851,148.213
C02642=1224.570,300.158,-66.960,-176.404,6.849,148.213
C02643=1224.575,299.910,-66.931,-176.407,6.847,148.214
C02644=1224.579,299.662,-66.902,-176.409,6.844,148.214
C02645=1224.584,299.414,-66.872,-176.411,6.842,148.214
C02646=1224.588,299.165,-66.844,-176.413,6.840,148.214
C02647=1224.592,298.917,-66.814,-176.416,6.836,148.214
C02648=1224.596,298.668,-66.785,-176.418,6.834,148.214
C02649=1224.601,298.420,-66.755,-176.420,6.832,148.214
C02650=1224.605,298.173,-66.726,-176.423,6.829,148.214
C02651=1224.610,297.924,-66.697,-176.426,6.827,148.214
C02652=1224.614,297.675,-66.668,-176.428,6.825,148.214
C02653=1224.618,297.427,-66.638,-176.430,6.822,148.214
C02654=1224.622,297.179,-66.609,-176.432,6.820,148.214
C02655=1224.627,296.931,-66.580,-176.435,6.817,148.214
C02656=1224.632,296.682,-66.551,-176.437,6.816,148.215
C02657=1224.636,296.434,-66.522,-176.440,6.812,148.215
C02658=1224.640,296.186,-66.492,-176.442,6.810,148.215
C02659=1224.644,295.938,-66.463,-176.444,6.808,148.215
C02660=1224.649,295.689,-66.434,-176.447,6.805,148.215
C02661=1224.653,295.441,-66.405,-176.449,6.803,148.215
C02662=1224.657,295.193,-66.376,-176.451,6.801,148.215
C02663=1224.661,294.944,-66.347,-176.454,6.798,148.215
C02664=1224.666,294.696,-66.318,-176.456,6.796,148.215
C02665=1224.670,294.448,-66.289,-176.459,6.794,148.215
C02666=1224.675,294.200,-66.260,-176.461,6.791,148.216
C02667=1224.679,293.951,-66.231,-176.464,6.788,148.216
C02668=1224.683,293.703,-66.201,-176.466,6.786,148.216
C02669=1224.688,293.455,-66.173,-176.468,6.784,148.216
C02670=1224.692,293.207,-66.144,-176.471,6.781,148.216
C02671=1224.696,292.958,-66.115,-176.473,6.779,148.216
C02672=1224.700,292.710,-66.086,-176.475,6.777,148.216
C02673=1224.705,292.462,-66.057,-176.478,6.774,148.216
C02674=1224.709,292.214,-66.029,-176.480,6.772,148.216
C02675=1224.713,291.965,-65.999,-176.482,6.770,148.216
C02676=1224.718,291.717,-65.971,-176.485,6.767,148.216
C02677=1224.722,291.469,-65.941,-176.487,6.764,148.216
C02678=1224.727,291.220,-65.913,-176.490,6.763,148.217
C02679=1224.730,290.972,-65.884,-176.492,6.760,148.217
C02680=1224.735,290.724,-65.855,-176.495,6.757,148.217
C02681=1224.740,290.476,-65.826,-176.497,6.755,148.217
C02682=1224.743,290.227,-65.798,-176.499,6.753,148.217
C02683=1224.748,289.979,-65.769,-176.501,6.751,148.217
C02684=1224.753,289.705,-65.737,-176.505,6.748,148.217
C02685=1224.758,289.431,-65.705,-176.507,6.745,148.217
C02686=1224.763,289.156,-65.674,-176.509,6.743,148.218
C02687=1224.767,288.882,-65.642,-176.513,6.740,148.218
C02688=1224.772,288.634,-65.613,-176.515,6.738,148.218
C02689=1224.776,288.386,-65.585,-176.517,6.736,148.218
C02690=1224.780,288.138,-65.555,-176.520,6.733,148.218
C02691=1224.785,287.889,-65.527,-176.522,6.731,148.218
C02692=1224.789,287.641,-65.499,-176.524,6.729,148.218
C02693=1224.793,287.393,-65.469,-176.527,6.727,148.219
C02694=1224.798,287.144,-65.441,-176.529,6.724,148.219
C02695=1224.802,286.896,-65.413,-176.531,6.721,148.219
C02696=1224.807,286.648,-65.384,-176.534,6.720,148.219
C02697=1224.811,286.399,-65.355,-176.537,6.717,148.219
C02698=1224.815,286.151,-65.327,-176.539,6.714,148.219
C02699=1224.820,285.903,-65.299,-176.541,6.712,148.219
C02700=1224.823,285.655,-65.270,-176.544,6.710,148.219
C02701=1224.829,285.406,-65.241,-176.547,6.707,148.220
C02702=1224.833,285.158,-65.213,-176.549,6.705,148.220
C02703=1224.837,284.909,-65.184,-176.551,6.703,148.220
C02704=1224.842,284.661,-65.156,-176.554,6.701,148.220
C02705=1224.845,284.413,-65.127,-176.556,6.698,148.220
C02706=1224.850,284.165,-65.099,-176.558,6.696,148.220
C02707=1224.854,283.916,-65.071,-176.561,6.694,148.220
C02708=1224.859,283.667,-65.042,-176.563,6.692,148.220
C02709=1224.863,283.419,-65.014,-176.566,6.689,148.220
C02710=1224.867,283.170,-64.985,-176.568,6.687,148.221
C02711=1224.872,282.923,-64.956,-176.570,6.685,148.221
C02712=1224.876,282.674,-64.928,-176.573,6.683,148.221
C02713=1224.881,282.426,-64.900,-176.576,6.680,148.221
C02714=1224.885,282.177,-64.872,-176.578,6.677,148.221
C02715=1224.890,281.929,-64.843,-176.580,6.676,148.222
C02716=1224.894,281.681,-64.815,-176.583,6.673,148.222
C02717=1224.898,281.433,-64.787,-176.585,6.671,148.222
C02718=1224.903,281.184,-64.759,-176.588,6.668,148.222
C02719=1224.907,280.936,-64.731,-176.590,6.666,148.222
C02720=1224.911,280.687,-64.702,-176.592,6.664,148.222
C02721=1224.916,280.439,-64.674,-176.595,6.662,148.222
C02722=1224.920,280.190,-64.646,-176.598,6.659,148.223
C02723=1224.925,279.943,-64.618,-176.600,6.657,148.223
C02724=1224.928,279.694,-64.590,-176.602,6.655,148.223
C02725=1224.933,279.446,-64.561,-176.605,6.653,148.223
C02726=1224.937,279.197,-64.533,-176.607,6.650,148.223
C02727=1224.942,278.949,-64.505,-176.610,6.648,148.223
C02728=1224.946,278.700,-64.477,-176.612,6.646,148.223
C02729=1224.950,278.453,-64.449,-176.615,6.644,148.224
C02730=1224.955,278.204,-64.420,-176.617,6.642,148.224
C02731=1224.959,277.956,-64.392,-176.620,6.639,148.224
C02732=1224.963,277.707,-64.365,-176.622,6.637,148.224
C02733=1224.968,277.458,-64.337,-176.624,6.635,148.224
C02734=1224.972,277.210,-64.308,-176.627,6.633,148.224
C02735=1224.977,276.962,-64.280,-176.629,6.631,148.224
C02736=1224.981,276.713,-64.252,-176.632,6.628,148.225
C02737=1224.985,276.465,-64.224,-176.634,6.626,148.225
C02738=1224.990,276.217,-64.197,-176.637,6.624,148.225
C02739=1224.994,275.968,-64.168,-176.639,6.622,148.225
C02740=1224.999,275.720,-64.141,-176.641,6.620,148.225
C02741=1225.002,275.471,-64.112,-176.644,6.617,148.225
C02742=1225.008,275.223,-64.084,-176.647,6.615,148.226
C02743=1225.012,274.974,-64.057,-176.649,6.613,148.226
C02744=1225.016,274.726,-64.029,-176.651,6.611,148.226
C02745=1225.020,274.478,-64.001,-176.653,6.608,148.226
C02746=1225.025,274.229,-63.972,-176.657,6.606,148.226
C02747=1225.029,273.981,-63.945,-176.659,6.603,148.227
C02748=1225.033,273.732,-63.917,-176.661,6.602,148.227
C02749=1225.038,273.484,-63.889,-176.663,6.599,148.227
C02750=1225.043,273.236,-63.862,-176.666,6.597,148.227
C02751=1225.047,272.987,-63.834,-176.669,6.594,148.227
C02752=1225.051,272.739,-63.806,-176.671,6.593,148.228
C02753=1225.056,272.491,-63.779,-176.673,6.590,148.228
C02754=1225.059,272.242,-63.751,-176.676,6.588,148.228
C02755=1225.065,271.994,-63.722,-176.678,6.586,148.228
C02756=1225.069,271.745,-63.695,-176.681,6.584,148.228
C02757=1225.073,271.497,-63.667,-176.683,6.581,148.228
C02758=1225.078,271.248,-63.640,-176.686,6.579,148.229
C02759=1225.082,271.000,-63.612,-176.688,6.577,148.229
C02760=1225.086,270.751,-63.585,-176.691,6.575,148.229
C02761=1225.091,270.503,-63.556,-176.693,6.573,148.229
C02762=1225.095,270.255,-63.529,-176.696,6.570,148.229
C02763=1225.100,270.006,-63.501,-176.698,6.568,148.229
C02764=1225.104,269.758,-63.473,-176.701,6.566,148.230
C02765=1225.109,269.510,-63.446,-176.703,6.564,148.230
C02766=1225.112,269.261,-63.418,-176.706,6.562,148.230
C02767=1225.117,269.013,-63.391,-176.708,6.560,148.230
C02768=1225.121,268.765,-63.363,-176.711,6.557,148.230
C02769=1225.125,268.515,-63.336,-176.713,6.555,148.231
C02770=1225.131,268.267,-63.308,-176.716,6.553,148.231
C02771=1225.135,268.019,-63.281,-176.718,6.551,148.231
C02772=1225.140,267.770,-63.253,-176.720,6.549,148.231
C02773=1225.144,267.522,-63.225,-176.723,6.547,148.231
C02774=1225.148,267.273,-63.198,-176.725,6.545,148.232
C02775=1225.153,267.025,-63.171,-176.728,6.542,148.232
C02776=1225.157,266.777,-63.143,-176.731,6.540,148.232
C02777=1225.161,266.528,-63.116,-176.733,6.538,148.232
C02778=1225.166,266.280,-63.088,-176.735,6.536,148.232
C02779=1225.170,266.031,-63.061,-176.738,6.534,148.232
C02780=1225.175,265.783,-63.034,-176.740,6.532,148.233
C02781=1225.179,265.534,-63.006,-176.743,6.530,148.233
C02782=1225.183,265.286,-62.979,-176.745,6.527,148.233
C02783=1225.188,265.037,-62.952,-176.748,6.525,148.233
C02784=1225.193,264.789,-62.925,-176.750,6.523,148.233
C02785=1225.196,264.540,-62.897,-176.753,6.521,148.234
C02786=1225.201,264.292,-62.870,-176.755,6.519,148.234
C02787=1225.206,264.043,-62.842,-176.758,6.517,148.234
C02788=1225.210,263.771,-62.813,-176.761,6.514,148.234
C02789=1225.215,263.498,-62.782,-176.763,6.513,148.235
C02790=1225.220,263.226,-62.753,-176.766,6.510,148.235
C02791=1225.225,262.954,-62.723,-176.769,6.508,148.235
C02792=1225.229,262.704,-62.696,-176.771,6.506,148.235
C02793=1225.233,262.456,-62.669,-176.774,6.504,148.236
C02794=1225.238,262.207,-62.641,-176.776,6.502,148.236
C02795=1225.243,261.959,-62.614,-176.778,6.500,148.236
C02796=1225.247,261.710,-62.587,-176.781,6.497,148.236
C02797=1225.251,261.462,-62.559,-176.784,6.495,148.236
C02798=1225.256,261.213,-62.532,-176.786,6.493,148.237
C02799=1225.260,260.965,-62.505,-176.789,6.491,148.237
C02800=1225.264,260.717,-62.479,-176.791,6.489,148.237
C02801=1225.269,260.468,-62.452,-176.794,6.487,148.237
C02802=1225.273,260.220,-62.425,-176.796,6.485,148.237
C02803=1225.278,259.971,-62.397,-176.798,6.483,148.238
C02804=1225.282,259.722,-62.370,-176.801,6.481,148.238
C02805=1225.287,259.474,-62.343,-176.804,6.478,148.238
C02806=1225.291,259.225,-62.316,-176.806,6.476,148.238
C02807=1225.295,258.977,-62.289,-176.808,6.474,148.238
C02808=1225.300,258.728,-62.262,-176.811,6.472,148.239
C02809=1225.305,258.480,-62.235,-176.814,6.470,148.239
C02810=1225.309,258.232,-62.209,-176.816,6.468,148.239
C02811=1225.313,257.983,-62.182,-176.818,6.466,148.239
C02812=1225.318,257.735,-62.155,-176.821,6.464,148.240
C02813=1225.322,257.485,-62.127,-176.823,6.462,148.240
C02814=1225.326,257.237,-62.101,-176.826,6.460,148.240
C02815=1225.331,256.989,-62.074,-176.829,6.457,148.240
C02816=1225.335,256.740,-62.047,-176.831,6.455,148.240
C02817=1225.340,256.492,-62.020,-176.834,6.453,148.241
C02818=1225.344,256.244,-61.993,-176.836,6.451,148.241
C02819=1225.349,255.995,-61.966,-176.838,6.449,148.241
C02820=1225.353,255.747,-61.939,-176.841,6.447,148.241
C02821=1225.357,255.498,-61.913,-176.844,6.445,148.242
C02822=1225.362,255.249,-61.886,-176.846,6.443,148.242
C02823=1225.367,255.001,-61.859,-176.848,6.441,148.242
C02824=1225.371,254.752,-61.832,-176.851,6.439,148.242
C02825=1225.375,254.504,-61.806,-176.854,6.438,148.243
C02826=1225.380,254.256,-61.779,-176.856,6.435,148.243
C02827=1225.384,254.007,-61.752,-176.858,6.434,148.243
C02828=1225.389,253.758,-61.726,-176.861,6.431,148.243
C02829=1225.393,253.510,-61.699,-176.864,6.429,148.244
C02830=1225.397,253.262,-61.672,-176.866,6.427,148.244
C02831=1225.402,253.013,-61.645,-176.869,6.425,148.244
C02832=1225.407,252.764,-61.619,-176.871,6.423,148.244
C02833=1225.411,252.516,-61.592,-176.874,6.421,148.245
C02834=1225.416,252.267,-61.565,-176.876,6.419,148.245
C02835=1225.420,252.019,-61.539,-176.879,6.417,148.245
C02836=1225.424,251.770,-61.513,-176.881,6.415,148.245
C02837=1225.429,251.522,-61.485,-176.884,6.413,148.246
C02838=1225.433,251.273,-61.459,-176.886,6.411,148.246
C02839=1225.438,251.024,-61.433,-176.888,6.409,148.246
C02840=1225.442,250.776,-61.406,-176.891,6.407,148.246
C02841=1225.447,250.528,-61.379,-176.893,6.405,148.247
C02842=1225.451,250.279,-61.353,-176.896,6.403,148.247
C02843=1225.455,250.030,-61.326,-176.898,6.401,148.247
C02844=1225.459,249.782,-61.300,-176.901,6.399,148.247
C02845=1225.464,249.533,-61.273,-176.903,6.397,148.248
C02846=1225.468,249.285,-61.247,-176.906,6.395,148.248
C02847=1225.473,249.036,-61.221,-176.909,6.392,148.248
C02848=1225.477,248.788,-61.194,-176.911,6.390,148.248
C02849=1225.482,248.538,-61.168,-176.914,6.389,148.249
C02850=1225.486,248.290,-61.141,-176.917,6.387,148.249
C02851=1225.491,248.042,-61.114,-176.919,6.384,148.249
C02852=1225.495,247.793,-61.089,-176.921,6.383,148.249
C02853=1225.500,247.544,-61.062,-176.924,6.381,148.250
C02854=1225.504,247.296,-61.036,-176.927,6.379,148.250
C02855=1225.509,247.048,-61.009,-176.929,6.377,148.250
C02856=1225.513,246.799,-60.983,-176.931,6.375,148.250
C02857=1225.518,246.551,-60.956,-176.934,6.373,148.251
C02858=1225.522,246.302,-60.931,-176.937,6.371,148.251
C02859=1225.526,246.053,-60.905,-176.939,6.369,148.251
C02860=1225.531,245.804,-60.878,-176.941,6.367,148.251
C02861=1225.535,245.556,-60.852,-176.944,6.365,148.252
C02862=1225.540,245.307,-60.825,-176.946,6.363,148.252
C02863=1225.544,245.058,-60.799,-176.949,6.361,148.252
C02864=1225.549,244.811,-60.773,-176.951,6.359,148.252
C02865=1225.554,244.562,-60.747,-176.954,6.357,148.253
C02866=1225.558,244.313,-60.721,-176.956,6.355,148.253
C02867=1225.562,244.065,-60.694,-176.959,6.354,148.253
C02868=1225.567,243.816,-60.668,-176.961,6.351,148.253
C02869=1225.571,243.567,-60.642,-176.964,6.349,148.254
C02870=1225.576,243.319,-60.616,-176.966,6.348,148.254
C02871=1225.580,243.070,-60.590,-176.969,6.346,148.254
C02872=1225.585,242.821,-60.564,-176.972,6.344,148.255
C02873=1225.589,242.573,-60.538,-176.974,6.342,148.255
C02874=1225.594,242.324,-60.511,-176.976,6.340,148.255
C02875=1225.598,242.075,-60.486,-176.979,6.338,148.255
C02876=1225.603,241.827,-60.460,-176.982,6.336,148.256
C02877=1225.607,241.579,-60.433,-176.984,6.334,148.256
C02878=1225.611,241.330,-60.407,-176.986,6.332,148.256
C02879=1225.616,241.081,-60.382,-176.989,6.330,148.256
C02880=1225.620,240.832,-60.356,-176.992,6.328,148.257
C02881=1225.625,240.584,-60.329,-176.994,6.326,148.257
C02882=1225.629,240.336,-60.303,-176.997,6.324,148.257
C02883=1225.634,240.087,-60.278,-176.999,6.322,148.257
C02884=1225.638,239.838,-60.252,-177.002,6.320,148.258
C02885=1225.643,239.589,-60.226,-177.004,6.318,148.258
C02886=1225.648,239.341,-60.200,-177.007,6.317,148.258
C02887=1225.652,239.093,-60.174,-177.009,6.315,148.259
C02888=1225.656,238.844,-60.148,-177.012,6.313,148.259
C02889=1225.661,238.595,-60.122,-177.014,6.311,148.259
C02890=1225.666,238.347,-60.096,-177.017,6.309,148.259
C02891=1225.670,238.098,-60.071,-177.019,6.307,148.260
C02892=1225.674,237.826,-60.042,-177.022,6.305,148.260
C02893=1225.679,237.555,-60.014,-177.025,6.303,148.260
C02894=1225.684,237.283,-59.986,-177.028,6.300,148.261
C02895=1225.689,237.012,-59.958,-177.030,6.299,148.261
C02896=1225.694,236.763,-59.933,-177.033,6.297,148.261
C02897=1225.698,236.515,-59.907,-177.036,6.295,148.262
C02898=1225.703,236.267,-59.880,-177.038,6.293,148.262
C02899=1225.707,236.018,-59.854,-177.040,6.291,148.262
C02900=1225.712,235.769,-59.829,-177.043,6.289,148.262
C02901=1225.716,235.520,-59.803,-177.046,6.287,148.263
C02902=1225.721,235.272,-59.778,-177.048,6.285,148.263
C02903=1225.725,235.023,-59.753,-177.051,6.283,148.263
C02904=1225.729,234.774,-59.727,-177.053,6.282,148.264
C02905=1225.734,234.526,-59.701,-177.056,6.280,148.264
C02906=1225.738,234.277,-59.676,-177.058,6.278,148.264
C02907=1225.743,234.028,-59.650,-177.060,6.276,148.264
C02908=1225.748,233.780,-59.624,-177.063,6.274,148.265
C02909=1225.752,233.531,-59.598,-177.066,6.273,148.265
C02910=1225.757,233.282,-59.572,-177.068,6.271,148.265
C02911=1225.762,233.034,-59.547,-177.071,6.269,148.266
C02912=1225.766,232.785,-59.521,-177.074,6.267,148.266
C02913=1225.770,232.536,-59.496,-177.076,6.265,148.266
C02914=1225.775,232.288,-59.471,-177.078,6.263,148.266
C02915=1225.779,232.039,-59.445,-177.081,6.261,148.267
C02916=1225.784,231.790,-59.419,-177.084,6.259,148.267
C02917=1225.788,231.542,-59.394,-177.086,6.257,148.267
C02918=1225.793,231.293,-59.368,-177.089,6.255,148.268
C02919=1225.798,231.045,-59.344,-177.091,6.254,148.268
C02920=1225.802,230.796,-59.318,-177.094,6.252,148.268
C02921=1225.806,230.547,-59.292,-177.097,6.250,148.269
C02922=1225.811,230.299,-59.267,-177.099,6.248,148.269
C02923=1225.815,230.050,-59.242,-177.101,6.247,148.269
C02924=1225.820,229.802,-59.217,-177.103,6.245,148.269
C02925=1225.824,229.553,-59.191,-177.106,6.243,148.270
C02926=1225.828,229.304,-59.165,-177.109,6.241,148.270
C02927=1225.833,229.055,-59.141,-177.111,6.239,148.270
C02928=1225.837,228.807,-59.115,-177.114,6.237,148.271
C02929=1225.842,228.559,-59.090,-177.117,6.235,148.271
C02930=1225.847,228.309,-59.064,-177.119,6.234,148.271
C02931=1225.851,228.060,-59.039,-177.122,6.232,148.272
C02932=1225.856,227.812,-59.013,-177.124,6.230,148.272
C02933=1225.860,227.563,-58.988,-177.127,6.228,148.272
C02934=1225.864,227.315,-58.964,-177.129,6.226,148.272
C02935=1225.869,227.066,-58.938,-177.132,6.224,148.273
C02936=1225.874,226.817,-58.913,-177.134,6.222,148.273
C02937=1225.878,226.569,-58.887,-177.137,6.221,148.273
C02938=1225.883,226.320,-58.863,-177.139,6.219,148.274
C02939=1225.887,226.071,-58.837,-177.142,6.217,148.274
C02940=1225.892,225.823,-58.813,-177.144,6.215,148.274
C02941=1225.896,225.574,-58.787,-177.147,6.214,148.275
C02942=1225.901,225.326,-58.762,-177.150,6.212,148.275
C02943=1225.905,225.076,-58.737,-177.152,6.210,148.275
C02944=1225.910,224.828,-58.711,-177.155,6.208,148.276
C02945=1225.915,224.579,-58.686,-177.158,6.206,148.276
C02946=1225.919,224.331,-58.661,-177.160,6.204,148.276
C02947=1225.923,224.082,-58.636,-177.163,6.202,148.277
C02948=1225.928,223.834,-58.611,-177.165,6.201,148.277
C02949=1225.933,223.584,-58.586,-177.167,6.199,148.277
C02950=1225.937,223.336,-58.562,-177.170,6.197,148.277
C02951=1225.941,223.087,-58.536,-177.172,6.195,148.278
C02952=1225.946,222.838,-58.512,-177.175,6.194,148.278
C02953=1225.951,222.589,-58.486,-177.177,6.192,148.278
C02954=1225.955,222.341,-58.462,-177.180,6.190,148.279
C02955=1225.959,222.092,-58.436,-177.183,6.188,148.279
C02956=1225.964,221.843,-58.411,-177.185,6.186,148.279
C02957=1225.968,221.594,-58.387,-177.188,6.184,148.280
C02958=1225.973,221.346,-58.361,-177.190,6.183,148.280
C02959=1225.978,221.097,-58.336,-177.193,6.181,148.280
C02960=1225.982,220.848,-58.312,-177.195,6.179,148.281
C02961=1225.987,220.600,-58.287,-177.198,6.178,148.281
C02962=1225.991,220.351,-58.262,-177.201,6.176,148.281
C02963=1225.996,220.102,-58.238,-177.203,6.174,148.282
C02964=1226.000,219.854,-58.212,-177.206,6.172,148.282
C02965=1226.005,219.605,-58.187,-177.208,6.170,148.282
C02966=1226.009,219.356,-58.163,-177.211,6.168,148.283
C02967=1226.014,219.108,-58.138,-177.214,6.166,148.283
C02968=1226.019,218.859,-58.113,-177.216,6.165,148.283
C02969=1226.023,218.610,-58.088,-177.218,6.164,148.284
C02970=1226.028,218.361,-58.064,-177.221,6.162,148.284
C02971=1226.031,218.113,-58.039,-177.224,6.160,148.284
C02972=1226.036,217.864,-58.014,-177.226,6.158,148.285
C02973=1226.042,217.615,-57.989,-177.229,6.156,148.285
C02974=1226.045,217.366,-57.965,-177.232,6.154,148.285
C02975=1226.050,217.117,-57.940,-177.234,6.152,148.286
C02976=1226.054,216.869,-57.915,-177.236,6.151,148.286
C02977=1226.059,216.620,-57.890,-177.239,6.149,148.286
C02978=1226.064,216.371,-57.866,-177.242,6.148,148.287
C02979=1226.068,216.122,-57.841,-177.244,6.146,148.287
C02980=1226.073,215.874,-57.817,-177.247,6.144,148.287
C02981=1226.078,215.625,-57.793,-177.249,6.142,148.288
C02982=1226.082,215.376,-57.768,-177.252,6.140,148.288
C02983=1226.086,215.127,-57.743,-177.255,6.138,148.288
C02984=1226.091,214.879,-57.718,-177.257,6.137,148.289
C02985=1226.095,214.630,-57.694,-177.259,6.135,148.289
C02986=1226.100,214.381,-57.669,-177.262,6.134,148.289
C02987=1226.105,214.133,-57.645,-177.265,6.132,148.290
C02988=1226.109,213.884,-57.620,-177.267,6.130,148.290
C02989=1226.114,213.635,-57.596,-177.270,6.128,148.290
C02990=1226.119,213.386,-57.571,-177.273,6.126,148.291
C02991=1226.123,213.138,-57.547,-177.275,6.124,148.291
C02992=1226.128,212.889,-57.522,-177.277,6.123,148.291
C02993=1226.132,212.640,-57.498,-177.280,6.121,148.292
C02994=1226.136,212.392,-57.474,-177.282,6.120,148.292
C02995=1226.141,212.142,-57.449,-177.285,6.118,148.292
C02996=1226.146,211.872,-57.422,-177.288,6.116,148.293
C02997=1226.151,211.602,-57.397,-177.291,6.114,148.293
C02998=1226.156,211.331,-57.370,-177.294,6.112,148.294
C02999=1226.160,211.061,-57.343,-177.296,6.111,148.294
C03000=1226.165,210.812,-57.319,-177.299,6.109,148.294
C03001=1226.170,210.563,-57.294,-177.301,6.107,148.295
C03002=1226.174,210.315,-57.270,-177.304,6.105,148.295
C03003=1226.179,210.065,-57.246,-177.307,6.103,148.295
C03004=1226.184,209.817,-57.222,-177.309,6.101,148.296
C03005=1226.188,209.568,-57.198,-177.311,6.100,148.296
C03006=1226.193,209.319,-57.173,-177.315,6.099,148.297
C03007=1226.198,209.071,-57.149,-177.317,6.097,148.297
C03008=1226.201,208.822,-57.124,-177.320,6.095,148.297
C03009=1226.207,208.573,-57.100,-177.322,6.093,148.298
C03010=1226.211,208.324,-57.076,-177.325,6.091,148.298
C03011=1226.216,208.076,-57.052,-177.327,6.090,148.298
C03012=1226.220,207.826,-57.027,-177.330,6.088,148.299
C03013=1226.224,207.578,-57.003,-177.332,6.087,148.299
C03014=1226.229,207.329,-56.980,-177.335,6.085,148.299
C03015=1226.234,207.080,-56.955,-177.338,6.083,148.300
C03016=1226.239,206.832,-56.931,-177.340,6.082,148.300
C03017=1226.243,206.583,-56.907,-177.342,6.080,148.300
C03018=1226.247,206.334,-56.883,-177.345,6.078,148.301
C03019=1226.252,206.085,-56.859,-177.348,6.076,148.301
C03020=1226.257,205.836,-56.835,-177.350,6.074,148.301
C03021=1226.261,205.587,-56.811,-177.352,6.073,148.302
C03022=1226.266,205.339,-56.787,-177.355,6.072,148.302
C03023=1226.270,205.090,-56.762,-177.358,6.070,148.303
C03024=1226.275,204.841,-56.739,-177.361,6.068,148.303
C03025=1226.279,204.592,-56.715,-177.363,6.066,148.303
C03026=1226.284,204.344,-56.691,-177.366,6.064,148.304
C03027=1226.289,204.095,-56.667,-177.368,6.063,148.304
C03028=1226.294,203.846,-56.643,-177.371,6.062,148.304
C03029=1226.298,203.598,-56.618,-177.373,6.060,148.305
C03030=1226.302,203.348,-56.595,-177.376,6.058,148.305
C03031=1226.307,203.099,-56.571,-177.378,6.057,148.305
C03032=1226.311,202.850,-56.547,-177.381,6.055,148.306
C03033=1226.316,202.602,-56.523,-177.384,6.054,148.306
C03034=1226.321,202.353,-56.499,-177.386,6.052,148.307
C03035=1226.325,202.104,-56.475,-177.389,6.050,148.307
C03036=1226.330,201.856,-56.451,-177.391,6.049,148.307
C03037=1226.335,201.607,-56.428,-177.394,6.047,148.308
C03038=1226.339,201.358,-56.404,-177.396,6.045,148.308
C03039=1226.343,201.109,-56.380,-177.399,6.043,148.308
C03040=1226.347,200.860,-56.356,-177.402,6.041,148.309
C03041=1226.352,200.611,-56.333,-177.404,6.040,148.309
C03042=1226.357,200.362,-56.308,-177.406,6.039,148.309
C03043=1226.362,200.113,-56.285,-177.410,6.037,148.310
C03044=1226.367,199.864,-56.261,-177.412,6.035,148.310
C03045=1226.371,199.616,-56.237,-177.414,6.034,148.311
C03046=1226.376,199.367,-56.214,-177.417,6.032,148.311
C03047=1226.380,199.119,-56.190,-177.420,6.030,148.311
C03048=1226.385,198.870,-56.166,-177.422,6.029,148.312
C03049=1226.389,198.621,-56.142,-177.424,6.028,148.312
C03050=1226.394,198.372,-56.119,-177.427,6.026,148.312
C03051=1226.399,198.123,-56.096,-177.430,6.024,148.313
C03052=1226.403,197.875,-56.071,-177.433,6.022,148.313
C03053=1226.408,197.626,-56.048,-177.435,6.021,148.314
C03054=1226.412,197.377,-56.025,-177.437,6.019,148.314
C03055=1226.417,197.128,-56.001,-177.440,6.018,148.314
C03056=1226.422,196.879,-55.977,-177.443,6.016,148.315
C03057=1226.426,196.630,-55.954,-177.445,6.015,148.315
C03058=1226.431,196.382,-55.930,-177.447,6.013,148.315
C03059=1226.435,196.133,-55.906,-177.451,6.011,148.316
C03060=1226.440,195.884,-55.883,-177.453,6.010,148.316
C03061=1226.445,195.635,-55.860,-177.455,6.009,148.317
C03062=1226.449,195.386,-55.836,-177.458,6.007,148.317
C03063=1226.454,195.137,-55.812,-177.461,6.005,148.317
C03064=1226.459,194.888,-55.789,-177.463,6.003,148.318
C03065=1226.463,194.639,-55.766,-177.465,6.002,148.318
C03066=1226.468,194.391,-55.742,-177.468,6.000,148.319
C03067=1226.472,194.142,-55.718,-177.471,5.999,148.319
C03068=1226.477,193.893,-55.695,-177.474,5.997,148.319
C03069=1226.482,193.644,-55.671,-177.476,5.996,148.320
C03070=1226.486,193.395,-55.649,-177.478,5.994,148.320
C03071=1226.490,193.146,-55.625,-177.481,5.992,148.320
C03072=1226.495,192.897,-55.601,-177.484,5.990,148.321
C03073=1226.500,192.648,-55.578,-177.486,5.990,148.321
C03074=1226.504,192.399,-55.555,-177.489,5.988,148.322
C03075=1226.509,192.150,-55.531,-177.492,5.986,148.322
C03076=1226.514,191.901,-55.508,-177.494,5.985,148.322
C03077=1226.518,191.652,-55.484,-177.496,5.983,148.323
C03078=1226.522,191.404,-55.462,-177.499,5.981,148.323
C03079=1226.527,191.156,-55.438,-177.502,5.980,148.324
C03080=1226.532,190.907,-55.415,-177.504,5.979,148.324
C03081=1226.537,190.658,-55.391,-177.507,5.977,148.324
C03082=1226.541,190.409,-55.368,-177.509,5.975,148.325
C03083=1226.546,190.160,-55.345,-177.512,5.974,148.325
C03084=1226.550,189.911,-55.322,-177.514,5.972,148.326
C03085=1226.555,189.662,-55.298,-177.517,5.971,148.326
C03086=1226.559,189.413,-55.275,-177.519,5.970,148.326
C03087=1226.564,189.164,-55.252,-177.522,5.968,148.327
C03088=1226.569,188.915,-55.228,-177.525,5.966,148.327
C03089=1226.573,188.667,-55.206,-177.527,5.964,148.328
C03090=1226.578,188.418,-55.183,-177.529,5.963,148.328
C03091=1226.583,188.169,-55.159,-177.533,5.961,148.328
C03092=1226.587,187.920,-55.136,-177.535,5.960,148.329
C03093=1226.591,187.671,-55.113,-177.537,5.959,148.329
C03094=1226.596,187.422,-55.090,-177.540,5.957,148.330
C03095=1226.601,187.172,-55.067,-177.543,5.955,148.330
C03096=1226.606,186.924,-55.045,-177.545,5.954,148.331
C03097=1226.610,186.675,-55.021,-177.548,5.952,148.331
C03098=1226.615,186.426,-54.998,-177.550,5.951,148.331
C03099=1226.620,186.177,-54.975,-177.553,5.950,148.332
C03100=1226.624,185.908,-54.950,-177.556,5.948,148.332
C03101=1226.630,185.638,-54.925,-177.558,5.946,148.333
C03102=1226.635,185.368,-54.900,-177.561,5.944,148.333
C03103=1226.640,185.099,-54.876,-177.564,5.943,148.333
C03104=1226.644,184.850,-54.852,-177.567,5.941,148.334
C03105=1226.649,184.601,-54.829,-177.569,5.940,148.334
C03106=1226.653,184.352,-54.806,-177.571,5.938,148.335
C03107=1226.658,184.104,-54.783,-177.575,5.937,148.335
C03108=1226.663,183.854,-54.761,-177.577,5.936,148.335
C03109=1226.667,183.605,-54.738,-177.579,5.934,148.336
C03110=1226.672,183.356,-54.714,-177.582,5.932,148.336
C03111=1226.677,183.108,-54.692,-177.584,5.931,148.337
C03112=1226.682,182.859,-54.669,-177.587,5.929,148.337
C03113=1226.686,182.610,-54.646,-177.590,5.928,148.337
C03114=1226.690,182.361,-54.623,-177.592,5.927,148.338
C03115=1226.695,182.112,-54.600,-177.595,5.925,148.338
C03116=1226.700,181.863,-54.578,-177.598,5.923,148.339
C03117=1226.704,181.614,-54.555,-177.600,5.922,148.339
C03118=1226.708,181.365,-54.532,-177.602,5.920,148.340
C03119=1226.713,181.116,-54.509,-177.605,5.919,148.340
C03120=1226.719,180.867,-54.486,-177.607,5.918,148.340
C03121=1226.723,180.619,-54.464,-177.610,5.916,148.341
C03122=1226.728,180.369,-54.441,-177.613,5.914,148.341
C03123=1226.732,180.121,-54.419,-177.615,5.913,148.342
C03124=1226.737,179.872,-54.395,-177.618,5.911,148.342
C03125=1226.741,179.623,-54.373,-177.620,5.911,148.343
C03126=1226.746,179.374,-54.350,-177.623,5.909,148.343
C03127=1226.751,179.125,-54.328,-177.626,5.907,148.343
C03128=1226.755,178.876,-54.305,-177.628,5.906,148.344
C03129=1226.759,178.627,-54.282,-177.631,5.905,148.344
C03130=1226.765,178.378,-54.260,-177.634,5.903,148.345
C03131=1226.769,178.130,-54.237,-177.636,5.902,148.345
C03132=1226.774,177.880,-54.214,-177.638,5.900,148.345
C03133=1226.778,177.631,-54.192,-177.641,5.899,148.346
C03134=1226.784,177.382,-54.169,-177.643,5.897,148.346
C03135=1226.788,177.133,-54.147,-177.646,5.896,148.347
C03136=1226.792,176.884,-54.125,-177.648,5.895,148.347
C03137=1226.797,176.636,-54.102,-177.651,5.893,148.348
C03138=1226.801,176.386,-54.080,-177.654,5.891,148.348
C03139=1226.806,176.137,-54.056,-177.656,5.890,148.348
C03140=1226.811,175.889,-54.034,-177.659,5.888,148.349
C03141=1226.816,175.640,-54.011,-177.661,5.888,148.349
C03142=1226.821,175.391,-53.989,-177.664,5.886,148.350
C03143=1226.825,175.142,-53.967,-177.667,5.884,148.350
C03144=1226.829,174.893,-53.944,-177.669,5.883,148.350
C03145=1226.834,174.644,-53.922,-177.672,5.881,148.351
C03146=1226.838,174.395,-53.900,-177.674,5.880,148.351
C03147=1226.843,174.146,-53.877,-177.677,5.879,148.352
C03148=1226.848,173.897,-53.855,-177.679,5.877,148.352
C03149=1226.853,173.648,-53.832,-177.682,5.876,148.353
C03150=1226.858,173.399,-53.810,-177.685,5.874,148.353
C03151=1226.862,173.151,-53.787,-177.687,5.873,148.353
C03152=1226.867,172.901,-53.765,-177.690,5.872,148.354
C03153=1226.872,172.652,-53.743,-177.692,5.870,148.354
C03154=1226.876,172.403,-53.721,-177.694,5.869,148.355
C03155=1226.881,172.155,-53.698,-177.697,5.867,148.355
C03156=1226.885,171.905,-53.676,-177.700,5.866,148.356
C03157=1226.890,171.656,-53.654,-177.702,5.865,148.356
C03158=1226.894,171.408,-53.632,-177.705,5.863,148.356
C03159=1226.899,171.158,-53.609,-177.708,5.862,148.357
C03160=1226.904,170.910,-53.587,-177.710,5.860,148.357
C03161=1226.908,170.660,-53.565,-177.712,5.859,148.358
C03162=1226.914,170.412,-53.542,-177.715,5.857,148.358
C03163=1226.918,170.163,-53.520,-177.718,5.856,148.359
C03164=1226.922,169.913,-53.498,-177.720,5.855,148.359
C03165=1226.927,169.665,-53.476,-177.723,5.853,148.360
C03166=1226.932,169.416,-53.453,-177.726,5.852,148.360
C03167=1226.937,169.167,-53.431,-177.728,5.851,148.361
C03168=1226.941,168.918,-53.409,-177.730,5.850,148.361
C03169=1226.946,168.669,-53.388,-177.733,5.848,148.361
C03170=1226.951,168.419,-53.365,-177.736,5.846,148.362
C03171=1226.956,168.171,-53.343,-177.738,5.845,148.362
C03172=1226.960,167.921,-53.321,-177.741,5.844,148.363
C03173=1226.965,167.673,-53.299,-177.743,5.843,148.363
C03174=1226.969,167.424,-53.277,-177.746,5.841,148.364
C03175=1226.974,167.175,-53.255,-177.748,5.840,148.364
C03176=1226.979,166.926,-53.233,-177.751,5.839,148.365
C03177=1226.984,166.677,-53.211,-177.753,5.838,148.365
C03178=1226.988,166.428,-53.189,-177.756,5.836,148.365
C03179=1226.993,166.179,-53.167,-177.759,5.834,148.366
C03180=1226.997,165.930,-53.145,-177.761,5.833,148.366
C03181=1227.002,165.681,-53.123,-177.764,5.831,148.367
C03182=1227.007,165.432,-53.101,-177.767,5.831,148.367
C03183=1227.012,165.183,-53.079,-177.769,5.829,148.368
C03184=1227.016,164.934,-53.057,-177.771,5.828,148.368
C03185=1227.021,164.685,-53.035,-177.774,5.826,148.369
C03186=1227.025,164.436,-53.013,-177.777,5.825,148.369
C03187=1227.030,164.187,-52.992,-177.779,5.824,148.369
C03188=1227.035,163.938,-52.970,-177.782,5.823,148.370
C03189=1227.039,163.689,-52.948,-177.784,5.821,148.370
C03190=1227.044,163.440,-52.926,-177.787,5.819,148.371
C03191=1227.048,163.191,-52.904,-177.790,5.819,148.371
C03192=1227.053,162.942,-52.882,-177.792,5.817,148.372
C03193=1227.058,162.693,-52.860,-177.794,5.816,148.372
C03194=1227.063,162.444,-52.838,-177.798,5.814,148.373
C03195=1227.067,162.195,-52.816,-177.800,5.813,148.373
C03196=1227.072,161.946,-52.794,-177.802,5.811,148.373
C03197=1227.077,161.697,-52.773,-177.805,5.811,148.374
C03198=1227.081,161.448,-52.751,-177.808,5.809,148.374
C03199=1227.086,161.199,-52.730,-177.810,5.808,148.375
C03200=1227.091,160.949,-52.708,-177.813,5.806,148.375
C03201=1227.096,160.701,-52.686,-177.815,5.805,148.376
C03202=1227.100,160.452,-52.664,-177.818,5.804,148.376
C03203=1227.105,160.203,-52.642,-177.820,5.803,148.377
C03204=1227.109,159.934,-52.619,-177.823,5.801,148.377
C03205=1227.115,159.665,-52.595,-177.826,5.800,148.378
C03206=1227.120,159.396,-52.572,-177.828,5.799,148.378
C03207=1227.125,159.127,-52.549,-177.831,5.797,148.379
C03208=1227.130,158.878,-52.528,-177.834,5.795,148.379
C03209=1227.134,158.629,-52.506,-177.836,5.795,148.380
C03210=1227.139,158.380,-52.484,-177.839,5.793,148.380
C03211=1227.144,158.131,-52.463,-177.841,5.792,148.380
C03212=1227.148,157.881,-52.441,-177.844,5.790,148.381
C03213=1227.153,157.633,-52.419,-177.847,5.789,148.381
C03214=1227.158,157.384,-52.398,-177.849,5.788,148.382
C03215=1227.163,157.134,-52.376,-177.852,5.787,148.382
C03216=1227.167,156.886,-52.354,-177.854,5.785,148.383
C03217=1227.172,156.637,-52.333,-177.857,5.784,148.383
C03218=1227.176,156.387,-52.312,-177.860,5.783,148.384
C03219=1227.181,156.139,-52.290,-177.862,5.782,148.384
C03220=1227.186,155.890,-52.269,-177.865,5.780,148.385
C03221=1227.191,155.640,-52.247,-177.867,5.779,148.385
C03222=1227.195,155.391,-52.226,-177.870,5.777,148.386
C03223=1227.200,155.143,-52.204,-177.872,5.777,148.386
C03224=1227.205,154.893,-52.183,-177.875,5.775,148.387
C03225=1227.209,154.644,-52.162,-177.878,5.774,148.387
C03226=1227.214,154.395,-52.141,-177.880,5.772,148.388
C03227=1227.219,154.147,-52.119,-177.882,5.771,148.388
C03228=1227.223,153.897,-52.097,-177.885,5.770,148.389
C03229=1227.228,153.648,-52.076,-177.888,5.769,148.389
C03230=1227.233,153.399,-52.054,-177.890,5.768,148.390
C03231=1227.237,153.150,-52.034,-177.893,5.766,148.390
C03232=1227.242,152.901,-52.012,-177.895,5.765,148.390
C03233=1227.247,152.652,-51.991,-177.898,5.764,148.391
C03234=1227.252,152.403,-51.969,-177.900,5.763,148.391
C03235=1227.257,152.153,-51.948,-177.903,5.762,148.392
C03236=1227.261,151.905,-51.927,-177.905,5.761,148.392
C03237=1227.266,151.656,-51.906,-177.908,5.759,148.393
C03238=1227.271,151.407,-51.884,-177.911,5.758,148.393
C03239=1227.275,151.157,-51.863,-177.913,5.756,148.394
C03240=1227.280,150.909,-51.842,-177.916,5.756,148.394
C03241=1227.285,150.659,-51.821,-177.919,5.754,148.395
C03242=1227.290,150.411,-51.799,-177.921,5.753,148.395
C03243=1227.295,150.161,-51.778,-177.923,5.752,148.396
C03244=1227.298,149.912,-51.757,-177.926,5.750,148.396
C03245=1227.303,149.663,-51.736,-177.929,5.750,148.397
C03246=1227.309,149.414,-51.715,-177.931,5.748,148.397
C03247=1227.313,149.166,-51.694,-177.933,5.747,148.397
C03248=1227.318,148.916,-51.673,-177.936,5.745,148.398
C03249=1227.322,148.667,-51.651,-177.939,5.744,148.398
C03250=1227.327,148.418,-51.630,-177.942,5.743,148.399
C03251=1227.332,148.169,-51.609,-177.944,5.742,148.399
C03252=1227.337,147.920,-51.588,-177.947,5.740,148.400
C03253=1227.341,147.671,-51.567,-177.949,5.739,148.400
C03254=1227.346,147.421,-51.546,-177.951,5.738,148.401
C03255=1227.351,147.173,-51.524,-177.954,5.737,148.401
C03256=1227.355,146.924,-51.504,-177.956,5.736,148.402
C03257=1227.360,146.674,-51.483,-177.960,5.735,148.402
C03258=1227.365,146.426,-51.461,-177.962,5.734,148.403
C03259=1227.369,146.177,-51.441,-177.965,5.732,148.403
C03260=1227.374,145.927,-51.419,-177.967,5.731,148.404
C03261=1227.378,145.678,-51.399,-177.969,5.730,148.404
C03262=1227.383,145.429,-51.377,-177.972,5.729,148.405
C03263=1227.389,145.180,-51.356,-177.974,5.728,148.405
C03264=1227.393,144.931,-51.336,-177.978,5.726,148.406
C03265=1227.398,144.682,-51.315,-177.980,5.725,148.406
C03266=1227.402,144.433,-51.294,-177.983,5.724,148.407
C03267=1227.407,144.184,-51.273,-177.985,5.723,148.407
C03268=1227.411,143.935,-51.252,-177.988,5.722,148.408
C03269=1227.416,143.685,-51.231,-177.990,5.720,148.408
C03270=1227.422,143.436,-51.210,-177.992,5.719,148.409
C03271=1227.426,143.188,-51.189,-177.995,5.718,148.409
C03272=1227.431,142.938,-51.168,-177.998,5.717,148.410
C03273=1227.435,142.690,-51.148,-178.000,5.716,148.410
C03274=1227.441,142.440,-51.127,-178.003,5.714,148.411
C03275=1227.445,142.191,-51.107,-178.005,5.714,148.411
C03276=1227.450,141.942,-51.086,-178.008,5.712,148.412
C03277=1227.455,141.693,-51.065,-178.011,5.711,148.412
C03278=1227.459,141.443,-51.044,-178.013,5.710,148.413
C03279=1227.463,141.195,-51.023,-178.016,5.709,148.413
C03280=1227.468,140.946,-51.002,-178.018,5.708,148.414
C03281=1227.473,140.697,-50.981,-178.021,5.706,148.414
C03282=1227.478,140.447,-50.961,-178.023,5.705,148.415
C03283=1227.483,140.198,-50.940,-178.025,5.704,148.415
C03284=1227.487,139.949,-50.920,-178.029,5.703,148.416
C03285=1227.492,139.700,-50.899,-178.031,5.702,148.416
C03286=1227.497,139.451,-50.878,-178.034,5.700,148.417
C03287=1227.502,139.202,-50.857,-178.036,5.699,148.417
C03288=1227.506,138.953,-50.837,-178.039,5.699,148.418
C03289=1227.511,138.704,-50.816,-178.041,5.697,148.418
C03290=1227.516,138.455,-50.796,-178.044,5.696,148.419
C03291=1227.521,138.206,-50.775,-178.047,5.695,148.419
C03292=1227.525,137.957,-50.754,-178.049,5.694,148.420
C03293=1227.530,137.708,-50.734,-178.051,5.693,148.420
C03294=1227.535,137.458,-50.713,-178.054,5.691,148.421
C03295=1227.539,137.209,-50.693,-178.056,5.690,148.421
C03296=1227.544,136.961,-50.672,-178.059,5.690,148.422
C03297=1227.549,136.711,-50.651,-178.062,5.688,148.422
C03298=1227.554,136.462,-50.632,-178.064,5.687,148.423
C03299=1227.559,136.212,-50.611,-178.067,5.686,148.423
C03300=1227.563,135.963,-50.590,-178.070,5.685,148.424
C03301=1227.568,135.715,-50.570,-178.072,5.684,148.424
C03302=1227.573,135.465,-50.549,-178.075,5.682,148.425
C03303=1227.577,135.216,-50.529,-178.077,5.682,148.425
C03304=1227.582,134.967,-50.508,-178.080,5.681,148.426
C03305=1227.587,134.718,-50.487,-178.082,5.679,148.426
C03306=1227.592,134.469,-50.468,-178.085,5.678,148.427
C03307=1227.596,134.220,-50.447,-178.087,5.677,148.427
C03308=1227.602,133.951,-50.425,-178.090,5.676,148.428
C03309=1227.607,133.682,-50.403,-178.093,5.675,148.429
C03310=1227.611,133.414,-50.381,-178.095,5.674,148.429
C03311=1227.617,133.145,-50.359,-178.099,5.672,148.430
C03312=1227.621,132.896,-50.339,-178.101,5.671,148.430
C03313=1227.627,132.646,-50.318,-178.103,5.670,148.431
C03314=1227.631,132.397,-50.298,-178.106,5.669,148.431
C03315=1227.636,132.149,-50.278,-178.109,5.668,148.432
C03316=1227.641,131.900,-50.258,-178.111,5.667,148.432
C03317=1227.646,131.650,-50.237,-178.114,5.666,148.433
C03318=1227.650,131.401,-50.217,-178.116,5.665,148.433
C03319=1227.655,131.152,-50.197,-178.119,5.664,148.434
C03320=1227.660,130.903,-50.177,-178.122,5.662,148.434
C03321=1227.664,130.654,-50.156,-178.124,5.662,148.435
C03322=1227.669,130.405,-50.135,-178.126,5.661,148.435
C03323=1227.674,130.155,-50.116,-178.129,5.659,148.436
C03324=1227.678,129.906,-50.095,-178.132,5.658,148.436
C03325=1227.684,129.657,-50.076,-178.134,5.657,148.437
C03326=1227.688,129.408,-50.056,-178.137,5.656,148.437
C03327=1227.693,129.159,-50.035,-178.139,5.655,148.438
C03328=1227.698,128.910,-50.015,-178.142,5.654,148.438
C03329=1227.702,128.661,-49.995,-178.144,5.653,148.439
C03330=1227.707,128.412,-49.974,-178.147,5.652,148.439
C03331=1227.712,128.162,-49.955,-178.149,5.651,148.440
C03332=1227.716,127.913,-49.934,-178.152,5.650,148.440
C03333=1227.722,127.664,-49.914,-178.154,5.649,148.441
C03334=1227.727,127.415,-49.894,-178.157,5.648,148.441
C03335=1227.731,127.166,-49.874,-178.160,5.646,148.442
C03336=1227.736,126.916,-49.854,-178.162,5.645,148.442
C03337=1227.740,126.667,-49.834,-178.165,5.645,148.443
C03338=1227.745,126.418,-49.814,-178.168,5.643,148.444
C03339=1227.750,126.170,-49.794,-178.170,5.642,148.444
C03340=1227.755,125.920,-49.774,-178.172,5.641,148.445
C03341=1227.759,125.671,-49.754,-178.175,5.641,148.445
C03342=1227.764,125.422,-49.734,-178.178,5.639,148.446
C03343=1227.769,125.172,-49.713,-178.180,5.638,148.446
C03344=1227.774,124.923,-49.694,-178.182,5.637,148.447
C03345=1227.779,124.675,-49.674,-178.185,5.636,148.447
C03346=1227.784,124.425,-49.654,-178.188,5.635,148.448
C03347=1227.788,124.176,-49.634,-178.190,5.634,148.448
C03348=1227.793,123.926,-49.614,-178.193,5.633,148.449
C03349=1227.798,123.678,-49.595,-178.196,5.632,148.449
C03350=1227.803,123.429,-49.574,-178.198,5.631,148.450
C03351=1227.807,123.179,-49.555,-178.200,5.630,148.450
C03352=1227.812,122.930,-49.534,-178.203,5.629,148.451
C03353=1227.817,122.681,-49.515,-178.206,5.628,148.452
C03354=1227.822,122.432,-49.495,-178.208,5.627,148.452
C03355=1227.826,122.183,-49.475,-178.211,5.626,148.453
C03356=1227.831,121.933,-49.455,-178.213,5.625,148.453
C03357=1227.835,121.684,-49.435,-178.216,5.624,148.454
C03358=1227.841,121.435,-49.416,-178.218,5.623,148.454
C03359=1227.846,121.186,-49.396,-178.221,5.622,148.455
C03360=1227.850,120.937,-49.376,-178.224,5.621,148.455
C03361=1227.855,120.687,-49.356,-178.226,5.620,148.456
C03362=1227.860,120.438,-49.337,-178.229,5.619,148.456
C03363=1227.865,120.189,-49.317,-178.231,5.618,148.457
C03364=1227.869,119.940,-49.297,-178.234,5.617,148.457
C03365=1227.875,119.691,-49.277,-178.236,5.616,148.458
C03366=1227.879,119.442,-49.258,-178.239,5.615,148.458
C03367=1227.883,119.193,-49.238,-178.242,5.614,148.459
C03368=1227.888,118.943,-49.218,-178.244,5.613,148.460
C03369=1227.893,118.694,-49.199,-178.247,5.612,148.460
C03370=1227.898,118.445,-49.179,-178.249,5.611,148.461
C03371=1227.902,118.196,-49.159,-178.252,5.610,148.461
C03372=1227.908,117.947,-49.140,-178.254,5.609,148.462
C03373=1227.912,117.697,-49.120,-178.257,5.608,148.462
C03374=1227.917,117.448,-49.100,-178.260,5.607,148.463
C03375=1227.922,117.199,-49.081,-178.262,5.606,148.463
C03376=1227.926,116.950,-49.061,-178.264,5.605,148.464
C03377=1227.931,116.701,-49.042,-178.267,5.604,148.464
C03378=1227.936,116.452,-49.022,-178.270,5.603,148.465
C03379=1227.941,116.202,-49.003,-178.272,5.602,148.466
C03380=1227.946,115.953,-48.983,-178.274,5.601,148.466
C03381=1227.951,115.704,-48.964,-178.278,5.600,148.467
C03382=1227.955,115.455,-48.945,-178.280,5.599,148.467
C03383=1227.960,115.206,-48.924,-178.282,5.598,148.468
C03384=1227.965,114.957,-48.905,-178.285,5.598,148.468
C03385=1227.970,114.707,-48.885,-178.288,5.596,148.469
C03386=1227.974,114.458,-48.866,-178.290,5.595,148.469
C03387=1227.980,114.209,-48.846,-178.293,5.595,148.470
C03388=1227.984,113.960,-48.827,-178.295,5.594,148.470
C03389=1227.989,113.711,-48.808,-178.298,5.592,148.471
C03390=1227.994,113.461,-48.788,-178.300,5.591,148.471
C03391=1227.999,113.212,-48.769,-178.303,5.591,148.472
C03392=1228.003,112.963,-48.750,-178.306,5.590,148.473
C03393=1228.008,112.713,-48.730,-178.308,5.588,148.473
C03394=1228.013,112.465,-48.711,-178.311,5.588,148.474
C03395=1228.018,112.215,-48.691,-178.313,5.587,148.474
C03396=1228.022,111.966,-48.672,-178.316,5.586,148.475
C03397=1228.027,111.717,-48.653,-178.318,5.585,148.475
C03398=1228.032,111.467,-48.633,-178.321,5.584,148.476
C03399=1228.037,111.218,-48.614,-178.323,5.583,148.476
C03400=1228.041,110.969,-48.595,-178.326,5.582,148.477
C03401=1228.046,110.720,-48.575,-178.328,5.581,148.478
C03402=1228.052,110.471,-48.556,-178.331,5.580,148.478
C03403=1228.056,110.221,-48.537,-178.334,5.579,148.479
C03404=1228.061,109.973,-48.518,-178.336,5.578,148.479
C03405=1228.066,109.723,-48.498,-178.339,5.578,148.480
C03406=1228.070,109.474,-48.479,-178.341,5.577,148.480
C03407=1228.075,109.225,-48.460,-178.344,5.575,148.481
C03408=1228.081,108.975,-48.441,-178.347,5.575,148.482
C03409=1228.085,108.726,-48.422,-178.349,5.574,148.482
C03410=1228.089,108.477,-48.402,-178.351,5.573,148.483
C03411=1228.095,108.228,-48.383,-178.355,5.572,148.483
C03412=1228.100,107.959,-48.362,-178.357,5.571,148.484
C03413=1228.104,107.691,-48.342,-178.359,5.570,148.484
C03414=1228.110,107.422,-48.322,-178.362,5.569,148.485
C03415=1228.115,107.154,-48.301,-178.365,5.568,148.486
C03416=1228.120,106.905,-48.281,-178.368,5.567,148.486
C03417=1228.124,106.656,-48.262,-178.370,5.566,148.487
C03418=1228.130,106.406,-48.244,-178.373,5.565,148.487
C03419=1228.135,106.157,-48.224,-178.376,5.564,148.488
C03420=1228.139,105.908,-48.205,-178.378,5.563,148.488
C03421=1228.144,105.659,-48.186,-178.380,5.563,148.489
C03422=1228.149,105.409,-48.168,-178.382,5.562,148.489
C03423=1228.154,105.160,-48.148,-178.386,5.560,148.490
C03424=1228.158,104.911,-48.129,-178.388,5.560,148.491
C03425=1228.163,104.662,-48.110,-178.390,5.559,148.491
C03426=1228.168,104.412,-48.091,-178.393,5.558,148.492
C03427=1228.173,104.163,-48.072,-178.396,5.558,148.492
C03428=1228.178,103.914,-48.053,-178.398,5.556,148.493
C03429=1228.182,103.665,-48.034,-178.401,5.555,148.493
C03430=1228.187,103.415,-48.015,-178.404,5.555,148.494
C03431=1228.192,103.166,-47.996,-178.406,5.554,148.494
C03432=1228.197,102.918,-47.977,-178.408,5.553,148.495
C03433=1228.202,102.668,-47.959,-178.411,5.552,148.496
C03434=1228.207,102.419,-47.939,-178.414,5.551,148.496
C03435=1228.211,102.170,-47.920,-178.416,5.550,148.497
C03436=1228.217,101.920,-47.902,-178.419,5.549,148.497
C03437=1228.221,101.671,-47.883,-178.421,5.548,148.498
C03438=1228.226,101.421,-47.864,-178.424,5.548,148.499
C03439=1228.231,101.173,-47.845,-178.427,5.546,148.499
C03440=1228.236,100.923,-47.826,-178.429,5.545,148.500
C03441=1228.240,100.674,-47.808,-178.431,5.545,148.500
C03442=1228.245,100.424,-47.788,-178.434,5.544,148.501
C03443=1228.250,100.175,-47.770,-178.436,5.543,148.501
C03444=1228.254,99.926,-47.751,-178.439,5.543,148.502
C03445=1228.260,99.677,-47.732,-178.442,5.541,148.503
C03446=1228.264,99.428,-47.714,-178.445,5.541,148.503
C03447=1228.269,99.178,-47.694,-178.447,5.540,148.504
C03448=1228.274,98.929,-47.676,-178.449,5.539,148.504
C03449=1228.279,98.681,-47.657,-178.452,5.538,148.505
C03450=1228.284,98.431,-47.638,-178.454,5.537,148.505
C03451=1228.288,98.182,-47.620,-178.457,5.536,148.506
C03452=1228.293,97.932,-47.601,-178.460,5.535,148.507
C03453=1228.298,97.683,-47.582,-178.462,5.534,148.507
C03454=1228.303,97.434,-47.564,-178.465,5.534,148.508
C03455=1228.308,97.184,-47.545,-178.467,5.533,148.508
C03456=1228.313,96.935,-47.527,-178.469,5.532,148.509
C03457=1228.318,96.686,-47.508,-178.472,5.532,148.509
C03458=1228.322,96.437,-47.489,-178.475,5.530,148.510
C03459=1228.327,96.187,-47.471,-178.478,5.530,148.511
C03460=1228.332,95.939,-47.452,-178.480,5.529,148.511
C03461=1228.337,95.689,-47.433,-178.483,5.528,148.512
C03462=1228.342,95.439,-47.415,-178.485,5.527,148.512
C03463=1228.347,95.191,-47.396,-178.487,5.527,148.513
C03464=1228.351,94.941,-47.378,-178.490,5.526,148.514
C03465=1228.356,94.692,-47.359,-178.493,5.525,148.514
C03466=1228.361,94.443,-47.341,-178.495,5.524,148.515
C03467=1228.366,94.193,-47.322,-178.498,5.523,148.515
C03468=1228.370,93.944,-47.303,-178.501,5.522,148.516
C03469=1228.375,93.695,-47.285,-178.503,5.522,148.517
C03470=1228.380,93.445,-47.266,-178.505,5.521,148.517
C03471=1228.385,93.196,-47.248,-178.508,5.520,148.518
C03472=1228.390,92.947,-47.230,-178.511,5.519,148.518
C03473=1228.394,92.697,-47.211,-178.513,5.518,148.519
C03474=1228.400,92.448,-47.192,-178.516,5.517,148.519
C03475=1228.405,92.199,-47.174,-178.518,5.517,148.520
C03476=1228.409,91.950,-47.156,-178.521,5.516,148.521
C03477=1228.414,91.700,-47.138,-178.523,5.515,148.521
C03478=1228.419,91.451,-47.119,-178.526,5.514,148.522
C03479=1228.424,91.202,-47.101,-178.528,5.514,148.522
C03480=1228.429,90.953,-47.083,-178.531,5.512,148.523
C03481=1228.433,90.703,-47.064,-178.534,5.511,148.523
C03482=1228.438,90.455,-47.046,-178.536,5.511,148.524
C03483=1228.443,90.205,-47.027,-178.539,5.510,148.525
C03484=1228.448,89.956,-47.009,-178.541,5.509,148.525
C03485=1228.453,89.706,-46.991,-178.544,5.509,148.526
C03486=1228.458,89.457,-46.973,-178.546,5.508,148.526
C03487=1228.462,89.208,-46.954,-178.549,5.507,148.527
C03488=1228.468,88.959,-46.935,-178.551,5.507,148.528
C03489=1228.472,88.709,-46.917,-178.554,5.505,148.528
C03490=1228.477,88.460,-46.899,-178.557,5.504,148.529
C03491=1228.482,88.211,-46.881,-178.560,5.504,148.529
C03492=1228.487,87.961,-46.863,-178.562,5.503,148.530
C03493=1228.492,87.713,-46.844,-178.564,5.502,148.531
C03494=1228.496,87.463,-46.826,-178.567,5.502,148.531
C03495=1228.501,87.213,-46.807,-178.569,5.501,148.532
C03496=1228.506,86.964,-46.790,-178.572,5.500,148.532
C03497=1228.511,86.715,-46.772,-178.574,5.500,148.533
C03498=1228.516,86.466,-46.754,-178.577,5.499,148.534
C03499=1228.521,86.216,-46.735,-178.580,5.497,148.534
C03500=1228.525,85.967,-46.717,-178.582,5.497,148.535
C03501=1228.530,85.718,-46.699,-178.585,5.496,148.535
C03502=1228.535,85.469,-46.681,-178.587,5.495,148.536
C03503=1228.540,85.219,-46.663,-178.590,5.494,148.536
C03504=1228.544,84.969,-46.645,-178.592,5.494,148.537
C03505=1228.550,84.720,-46.626,-178.595,5.493,148.538
C03506=1228.555,84.471,-46.608,-178.597,5.493,148.538
C03507=1228.560,84.222,-46.590,-178.600,5.492,148.539
C03508=1228.565,83.972,-46.572,-178.602,5.491,148.539
C03509=1228.570,83.723,-46.554,-178.605,5.491,148.540
C03510=1228.575,83.474,-46.536,-178.607,5.490,148.541
C03511=1228.579,83.224,-46.518,-178.610,5.488,148.541
C03512=1228.584,82.975,-46.500,-178.613,5.488,148.542
C03513=1228.589,82.726,-46.482,-178.615,5.487,148.542
C03514=1228.594,82.477,-46.464,-178.618,5.486,148.543
C03515=1228.599,82.228,-46.446,-178.620,5.485,148.544
C03516=1228.604,81.959,-46.427,-178.623,5.485,148.544
C03517=1228.609,81.691,-46.407,-178.625,5.484,148.545
C03518=1228.614,81.423,-46.388,-178.629,5.483,148.545
C03519=1228.619,81.154,-46.369,-178.631,5.482,148.546
C03520=1228.624,80.905,-46.351,-178.634,5.482,148.547
C03521=1228.629,80.656,-46.333,-178.636,5.481,148.547
C03522=1228.634,80.406,-46.315,-178.639,5.480,148.548
C03523=1228.639,80.157,-46.297,-178.641,5.479,148.549
C03524=1228.644,79.908,-46.279,-178.644,5.479,148.549
C03525=1228.648,79.658,-46.261,-178.647,5.478,148.550
C03526=1228.653,79.408,-46.244,-178.649,5.478,148.551
C03527=1228.658,79.159,-46.226,-178.652,5.477,148.551
C03528=1228.663,78.910,-46.208,-178.654,5.476,148.552
C03529=1228.668,78.661,-46.190,-178.657,5.476,148.552
C03530=1228.673,78.412,-46.172,-178.659,5.475,148.553
C03531=1228.678,78.162,-46.155,-178.662,5.474,148.554
C03532=1228.682,77.913,-46.137,-178.664,5.473,148.554
C03533=1228.687,77.664,-46.119,-178.667,5.472,148.555
C03534=1228.692,77.415,-46.101,-178.670,5.471,148.555
C03535=1228.697,77.165,-46.083,-178.672,5.471,148.556
C03536=1228.702,76.916,-46.066,-178.675,5.470,148.557
C03537=1228.707,76.666,-46.048,-178.677,5.469,148.557
C03538=1228.712,76.417,-46.030,-178.680,5.469,148.558
C03539=1228.717,76.168,-46.012,-178.682,5.468,148.558
C03540=1228.722,75.919,-45.995,-178.685,5.468,148.559
C03541=1228.727,75.669,-45.977,-178.688,5.467,148.560
C03542=1228.731,75.420,-45.959,-178.690,5.466,148.560
C03543=1228.737,75.170,-45.942,-178.692,5.465,148.561
C03544=1228.742,74.921,-45.924,-178.695,5.465,148.561
C03545=1228.746,74.672,-45.906,-178.698,5.464,148.562
C03546=1228.751,74.423,-45.890,-178.700,5.464,148.563
C03547=1228.756,74.173,-45.872,-178.702,5.463,148.563
C03548=1228.761,73.924,-45.854,-178.705,5.462,148.564
C03549=1228.766,73.675,-45.836,-178.708,5.461,148.565
C03550=1228.771,73.425,-45.818,-178.710,5.461,148.565
C03551=1228.775,73.176,-45.801,-178.713,5.460,148.566
C03552=1228.780,72.927,-45.784,-178.715,5.459,148.566
C03553=1228.785,72.678,-45.766,-178.718,5.459,148.567
C03554=1228.790,72.428,-45.748,-178.720,5.458,148.568
C03555=1228.795,72.179,-45.731,-178.723,5.458,148.568
C03556=1228.799,71.930,-45.713,-178.726,5.457,148.569
C03557=1228.805,71.680,-45.696,-178.728,5.456,148.569
C03558=1228.810,71.431,-45.678,-178.730,5.455,148.570
C03559=1228.814,71.181,-45.661,-178.733,5.455,148.571
C03560=1228.819,70.932,-45.643,-178.736,5.454,148.571
C03561=1228.824,70.682,-45.626,-178.738,5.454,148.572
C03562=1228.829,70.433,-45.608,-178.740,5.453,148.572
C03563=1228.834,70.184,-45.591,-178.744,5.451,148.573
C03564=1228.839,69.934,-45.573,-178.746,5.451,148.574
C03565=1228.844,69.685,-45.556,-178.749,5.450,148.574
C03566=1228.848,69.436,-45.539,-178.751,5.450,148.575
C03567=1228.853,69.186,-45.521,-178.754,5.449,148.575
C03568=1228.858,68.937,-45.503,-178.756,5.448,148.576
C03569=1228.863,68.687,-45.486,-178.759,5.448,148.577
C03570=1228.868,68.439,-45.469,-178.761,5.447,148.577
C03571=1228.873,68.189,-45.452,-178.764,5.446,148.578
C03572=1228.878,67.940,-45.434,-178.767,5.446,148.579
C03573=1228.883,67.690,-45.417,-178.769,5.445,148.579
C03574=1228.888,67.441,-45.400,-178.771,5.444,148.580
C03575=1228.892,67.192,-45.383,-178.774,5.444,148.581
C03576=1228.897,66.942,-45.365,-178.777,5.443,148.581
C03577=1228.902,66.693,-45.347,-178.779,5.442,148.582
C03578=1228.907,66.443,-45.331,-178.782,5.442,148.582
C03579=1228.912,66.194,-45.313,-178.784,5.441,148.583
C03580=1228.917,65.945,-45.296,-178.787,5.440,148.584
C03581=1228.922,65.695,-45.279,-178.789,5.440,148.584
C03582=1228.927,65.446,-45.261,-178.792,5.439,148.585
C03583=1228.931,65.197,-45.244,-178.795,5.439,148.586
C03584=1228.936,64.947,-45.227,-178.797,5.438,148.586
C03585=1228.941,64.698,-45.209,-178.799,5.438,148.587
C03586=1228.946,64.448,-45.193,-178.801,5.437,148.587
C03587=1228.952,64.199,-45.176,-178.804,5.437,148.588
C03588=1228.956,63.950,-45.158,-178.807,5.436,148.589
C03589=1228.961,63.701,-45.141,-178.809,5.436,148.589
C03590=1228.966,63.451,-45.124,-178.812,5.435,148.590
C03591=1228.971,63.201,-45.107,-178.814,5.434,148.590
C03592=1228.975,62.952,-45.090,-178.817,5.434,148.591
C03593=1228.981,62.703,-45.073,-178.819,5.433,148.592
C03594=1228.986,62.454,-45.055,-178.822,5.432,148.592
C03595=1228.990,62.204,-45.039,-178.825,5.432,148.593
C03596=1228.995,61.955,-45.021,-178.827,5.431,148.594
C03597=1229.000,61.705,-45.004,-178.829,5.430,148.594
C03598=1229.005,61.456,-44.987,-178.832,5.430,148.595
C03599=1229.010,61.207,-44.971,-178.835,5.429,148.596
C03600=1229.015,60.958,-44.953,-178.837,5.429,148.596
C03601=1229.020,60.708,-44.936,-178.840,5.428,148.597
C03602=1229.025,60.458,-44.919,-178.843,5.427,148.598
C03603=1229.029,60.209,-44.902,-178.845,5.426,148.598
C03604=1229.035,59.960,-44.885,-178.847,5.426,148.599
C03605=1229.040,59.710,-44.868,-178.850,5.425,148.599
C03606=1229.044,59.461,-44.851,-178.853,5.425,148.600
C03607=1229.049,59.212,-44.834,-178.855,5.424,148.601
C03608=1229.054,58.963,-44.818,-178.858,5.424,148.601
C03609=1229.059,58.713,-44.800,-178.861,5.423,148.602
C03610=1229.064,58.464,-44.784,-178.863,5.422,148.602
C03611=1229.069,58.214,-44.766,-178.865,5.421,148.603
C03612=1229.074,57.965,-44.750,-178.868,5.421,148.604
C03613=1229.079,57.715,-44.733,-178.871,5.420,148.604
C03614=1229.083,57.466,-44.715,-178.873,5.420,148.605
C03615=1229.088,57.217,-44.699,-178.876,5.419,148.606
C03616=1229.094,56.968,-44.682,-178.879,5.419,148.606
C03617=1229.098,56.718,-44.665,-178.880,5.418,148.607
C03618=1229.103,56.469,-44.648,-178.883,5.418,148.608
C03619=1229.108,56.219,-44.631,-178.885,5.417,148.608
C03620=1229.113,55.951,-44.613,-178.888,5.417,148.609
C03621=1229.119,55.682,-44.595,-178.891,5.415,148.610
C03622=1229.124,55.414,-44.578,-178.894,5.415,148.610
C03623=1229.129,55.145,-44.559,-178.897,5.415,148.611
C03624=1229.135,54.896,-44.543,-178.899,5.414,148.612
C03625=1229.139,54.647,-44.526,-178.902,5.413,148.612
C03626=1229.144,54.397,-44.509,-178.904,5.412,148.613
C03627=1229.149,54.148,-44.493,-178.907,5.412,148.614
C03628=1229.154,53.899,-44.476,-178.909,5.412,148.614
C03629=1229.159,53.649,-44.459,-178.912,5.412,148.615
C03630=1229.164,53.400,-44.442,-178.914,5.411,148.616
C03631=1229.169,53.151,-44.426,-178.917,5.410,148.616
C03632=1229.174,52.901,-44.408,-178.919,5.409,148.617
C03633=1229.178,52.651,-44.392,-178.922,5.409,148.617
C03634=1229.183,52.403,-44.375,-178.924,5.408,148.618
C03635=1229.189,52.153,-44.358,-178.927,5.408,148.619
C03636=1229.193,51.903,-44.341,-178.930,5.407,148.619
C03637=1229.198,51.654,-44.325,-178.932,5.407,148.620
C03638=1229.203,51.404,-44.309,-178.935,5.406,148.621
C03639=1229.208,51.155,-44.292,-178.938,5.405,148.621
C03640=1229.213,50.906,-44.276,-178.940,5.405,148.622
C03641=1229.218,50.656,-44.259,-178.942,5.404,148.622
C03642=1229.223,50.408,-44.243,-178.944,5.404,148.623
